Yaskawa INFORM job: DEMO_ROOF_UPPER_0625_3PAINT_59.JBI

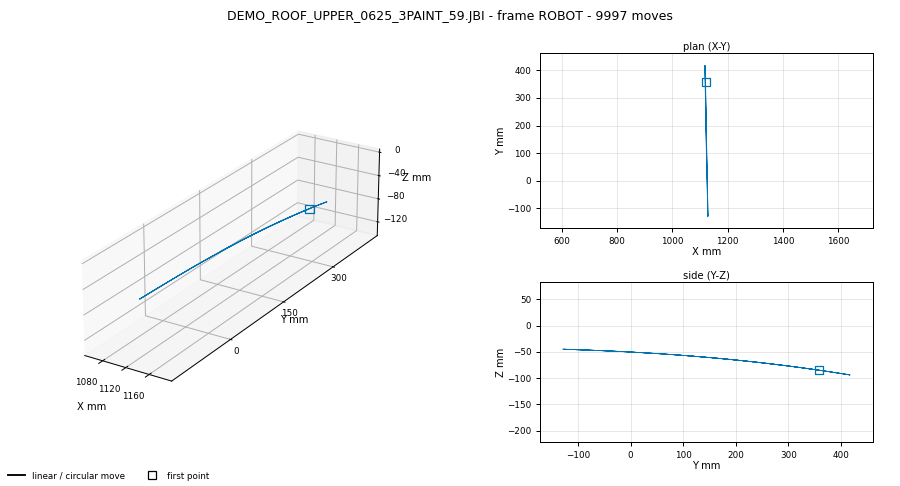
[picture p0: tool path of DEMO_ROOF_UPPER_0625_3PAINT_59.JBI in frame ROBOT, 9997 of 9997 moves have a stored position in this frame; points joined in program order, loops and branches not executed]
/JOB
//NAME DEMO_ROOF_UPPER_0625_3PAINT59
//POS
///NPOS 9997,0,0,0,0,0
///TOOL 0
///USER 0
///POSTYPE ROBOT
///RECTAN
///RCONF 1,0,0,0,0,0,0,0,0,0,0,0,0,0,0,0,0,0,0,0,0,0,0,0
C00000=1119.917,358.659,-84.729,-177.151,11.041,149.489
C00001=1119.921,358.412,-84.693,-177.154,11.038,149.489
C00002=1119.925,358.165,-84.658,-177.158,11.036,149.490
C00003=1119.929,357.918,-84.622,-177.161,11.033,149.490
C00004=1119.933,357.670,-84.586,-177.165,11.031,149.490
C00005=1119.936,357.423,-84.550,-177.168,11.029,149.490
C00006=1119.940,357.176,-84.514,-177.171,11.026,149.491
C00007=1119.944,356.928,-84.479,-177.175,11.024,149.491
C00008=1119.948,356.680,-84.443,-177.179,11.021,149.491
C00009=1119.952,356.433,-84.407,-177.182,11.019,149.491
C00010=1119.955,356.185,-84.372,-177.186,11.016,149.492
C00011=1119.959,355.938,-84.336,-177.189,11.014,149.492
C00012=1119.963,355.691,-84.301,-177.192,11.011,149.492
C00013=1119.967,355.444,-84.265,-177.196,11.009,149.492
C00014=1119.971,355.196,-84.229,-177.199,11.007,149.493
C00015=1119.975,354.948,-84.194,-177.203,11.004,149.493
C00016=1119.979,354.701,-84.158,-177.206,11.002,149.493
C00017=1119.982,354.453,-84.123,-177.209,10.999,149.493
C00018=1119.986,354.206,-84.087,-177.212,10.997,149.494
C00019=1119.990,353.959,-84.052,-177.217,10.994,149.494
C00020=1119.994,353.711,-84.016,-177.220,10.991,149.494
C00021=1119.997,353.464,-83.981,-177.223,10.989,149.494
C00022=1120.001,353.216,-83.945,-177.227,10.986,149.495
C00023=1120.006,352.969,-83.909,-177.230,10.984,149.495
C00024=1120.010,352.722,-83.874,-177.233,10.981,149.495
C00025=1120.013,352.474,-83.838,-177.237,10.979,149.495
C00026=1120.017,352.227,-83.803,-177.241,10.976,149.496
C00027=1120.021,351.979,-83.767,-177.244,10.974,149.496
C00028=1120.025,351.731,-83.732,-177.248,10.971,149.496
C00029=1120.029,351.484,-83.697,-177.251,10.969,149.496
C00030=1120.033,351.237,-83.662,-177.254,10.966,149.497
C00031=1120.036,350.989,-83.626,-177.258,10.964,149.497
C00032=1120.040,350.742,-83.591,-177.261,10.961,149.497
C00033=1120.045,350.494,-83.556,-177.265,10.958,149.497
C00034=1120.048,350.247,-83.521,-177.268,10.956,149.498
C00035=1120.052,349.999,-83.485,-177.272,10.953,149.498
C00036=1120.056,349.751,-83.450,-177.275,10.951,149.498
C00037=1120.059,349.505,-83.416,-177.279,10.948,149.498
C00038=1120.063,349.292,-83.385,-177.282,10.946,149.498
C00039=1120.066,349.080,-83.355,-177.284,10.944,149.499
C00040=1120.070,348.867,-83.325,-177.287,10.942,149.499
C00041=1120.073,348.655,-83.295,-177.290,10.940,149.499
C00042=1120.077,348.443,-83.265,-177.293,10.937,149.499
C00043=1120.079,348.230,-83.234,-177.296,10.935,149.499
C00044=1120.083,348.018,-83.204,-177.298,10.933,149.499
C00045=1120.086,347.805,-83.174,-177.301,10.931,149.500
C00046=1120.090,347.558,-83.139,-177.305,10.929,149.500
C00047=1120.095,347.310,-83.104,-177.307,10.926,149.500
C00048=1120.098,347.063,-83.069,-177.310,10.924,149.500
C00049=1120.101,346.815,-83.034,-177.313,10.922,149.500
C00050=1120.106,346.568,-82.999,-177.317,10.919,149.501
C00051=1120.110,346.320,-82.964,-177.320,10.917,149.501
C00052=1120.113,346.073,-82.929,-177.323,10.914,149.501
C00053=1120.118,345.825,-82.894,-177.327,10.912,149.501
C00054=1120.122,345.578,-82.859,-177.330,10.909,149.501
C00055=1120.125,345.331,-82.825,-177.333,10.907,149.502
C00056=1120.129,345.083,-82.789,-177.336,10.904,149.502
C00057=1120.133,344.835,-82.755,-177.340,10.902,149.502
C00058=1120.138,344.588,-82.720,-177.343,10.899,149.502
C00059=1120.141,344.340,-82.685,-177.346,10.897,149.503
C00060=1120.145,344.093,-82.651,-177.349,10.894,149.503
C00061=1120.149,343.846,-82.615,-177.352,10.891,149.503
C00062=1120.153,343.597,-82.580,-177.355,10.890,149.503
C00063=1120.157,343.350,-82.546,-177.358,10.887,149.503
C00064=1120.160,343.103,-82.511,-177.362,10.885,149.504
C00065=1120.165,342.855,-82.476,-177.365,10.882,149.504
C00066=1120.169,342.607,-82.442,-177.368,10.880,149.504
C00067=1120.173,342.360,-82.408,-177.371,10.877,149.504
C00068=1120.176,342.113,-82.372,-177.375,10.875,149.504
C00069=1120.180,341.865,-82.337,-177.378,10.872,149.505
C00070=1120.184,341.617,-82.304,-177.381,10.869,149.505
C00071=1120.188,341.369,-82.269,-177.384,10.867,149.505
C00072=1120.193,341.122,-82.234,-177.387,10.865,149.505
C00073=1120.195,340.875,-82.199,-177.391,10.862,149.505
C00074=1120.200,340.627,-82.165,-177.394,10.860,149.506
C00075=1120.204,340.379,-82.130,-177.397,10.857,149.506
C00076=1120.208,340.132,-82.096,-177.400,10.854,149.506
C00077=1120.212,339.884,-82.061,-177.403,10.853,149.506
C00078=1120.216,339.637,-82.027,-177.406,10.850,149.506
C00079=1120.220,339.389,-81.993,-177.410,10.848,149.507
C00080=1120.224,339.141,-81.958,-177.413,10.845,149.507
C00081=1120.227,338.894,-81.923,-177.416,10.843,149.507
C00082=1120.232,338.647,-81.889,-177.419,10.840,149.507
C00083=1120.235,338.399,-81.854,-177.422,10.838,149.507
C00084=1120.239,338.151,-81.820,-177.425,10.835,149.507
C00085=1120.243,337.904,-81.786,-177.429,10.832,149.508
C00086=1120.247,337.656,-81.751,-177.432,10.830,149.508
C00087=1120.251,337.409,-81.717,-177.435,10.827,149.508
C00088=1120.255,337.161,-81.683,-177.439,10.825,149.508
C00089=1120.259,336.914,-81.649,-177.442,10.822,149.508
C00090=1120.263,336.665,-81.615,-177.445,10.820,149.509
C00091=1120.267,336.418,-81.581,-177.448,10.818,149.509
C00092=1120.271,336.170,-81.546,-177.451,10.816,149.509
C00093=1120.275,335.923,-81.512,-177.454,10.813,149.509
C00094=1120.278,335.711,-81.482,-177.457,10.810,149.509
C00095=1120.282,335.498,-81.454,-177.459,10.808,149.509
C00096=1120.285,335.285,-81.424,-177.462,10.807,149.510
C00097=1120.289,335.073,-81.394,-177.465,10.804,149.510
C00098=1120.292,334.860,-81.365,-177.468,10.802,149.510
C00099=1120.295,334.648,-81.335,-177.471,10.800,149.510
C00100=1120.299,334.435,-81.306,-177.473,10.798,149.510
C00101=1120.302,334.223,-81.277,-177.476,10.796,149.510
C00102=1120.306,333.975,-81.243,-177.479,10.793,149.511
C00103=1120.310,333.727,-81.209,-177.482,10.791,149.511
C00104=1120.314,333.480,-81.175,-177.485,10.788,149.511
C00105=1120.318,333.233,-81.141,-177.488,10.786,149.511
C00106=1120.321,332.985,-81.107,-177.492,10.783,149.511
C00107=1120.326,332.737,-81.073,-177.495,10.781,149.512
C00108=1120.329,332.489,-81.039,-177.498,10.778,149.512
C00109=1120.333,332.242,-81.005,-177.501,10.776,149.512
C00110=1120.338,331.994,-80.971,-177.505,10.773,149.512
C00111=1120.341,331.746,-80.937,-177.508,10.771,149.512
C00112=1120.345,331.499,-80.903,-177.511,10.768,149.513
C00113=1120.350,331.251,-80.869,-177.514,10.766,149.513
C00114=1120.353,331.003,-80.835,-177.517,10.764,149.513
C00115=1120.357,330.755,-80.802,-177.520,10.761,149.513
C00116=1120.361,330.508,-80.768,-177.523,10.759,149.513
C00117=1120.366,330.261,-80.734,-177.526,10.756,149.514
C00118=1120.369,330.012,-80.700,-177.530,10.754,149.514
C00119=1120.373,329.765,-80.666,-177.533,10.751,149.514
C00120=1120.377,329.517,-80.633,-177.536,10.748,149.514
C00121=1120.381,329.269,-80.598,-177.539,10.746,149.514
C00122=1120.385,329.022,-80.565,-177.542,10.743,149.514
C00123=1120.389,328.774,-80.531,-177.546,10.741,149.515
C00124=1120.393,328.527,-80.498,-177.549,10.738,149.515
C00125=1120.397,328.279,-80.464,-177.552,10.736,149.515
C00126=1120.401,328.031,-80.430,-177.555,10.733,149.515
C00127=1120.406,327.783,-80.397,-177.558,10.731,149.516
C00128=1120.409,327.536,-80.363,-177.561,10.729,149.516
C00129=1120.413,327.288,-80.329,-177.564,10.726,149.516
C00130=1120.417,327.041,-80.296,-177.567,10.724,149.516
C00131=1120.421,326.793,-80.262,-177.571,10.721,149.516
C00132=1120.425,326.545,-80.229,-177.574,10.719,149.516
C00133=1120.429,326.297,-80.194,-177.577,10.716,149.517
C00134=1120.433,326.049,-80.161,-177.580,10.714,149.517
C00135=1120.437,325.801,-80.128,-177.583,10.711,149.517
C00136=1120.441,325.554,-80.094,-177.587,10.708,149.517
C00137=1120.445,325.307,-80.061,-177.590,10.706,149.517
C00138=1120.449,325.058,-80.028,-177.593,10.703,149.517
C00139=1120.453,324.810,-79.994,-177.596,10.701,149.518
C00140=1120.457,324.563,-79.961,-177.599,10.698,149.518
C00141=1120.461,324.316,-79.927,-177.602,10.696,149.518
C00142=1120.465,324.068,-79.894,-177.605,10.694,149.518
C00143=1120.469,323.820,-79.861,-177.608,10.691,149.519
C00144=1120.472,323.572,-79.827,-177.611,10.689,149.519
C00145=1120.477,323.325,-79.794,-177.615,10.686,149.519
C00146=1120.481,323.077,-79.761,-177.618,10.684,149.519
C00147=1120.485,322.829,-79.727,-177.621,10.681,149.519
C00148=1120.489,322.581,-79.694,-177.624,10.678,149.519
C00149=1120.493,322.334,-79.661,-177.628,10.676,149.520
C00150=1120.497,322.121,-79.632,-177.630,10.674,149.520
C00151=1120.499,321.908,-79.604,-177.633,10.671,149.520
C00152=1120.503,321.695,-79.575,-177.635,10.670,149.520
C00153=1120.507,321.483,-79.547,-177.638,10.668,149.520
C00154=1120.510,321.271,-79.518,-177.641,10.665,149.520
C00155=1120.513,321.058,-79.489,-177.643,10.663,149.521
C00156=1120.516,320.845,-79.461,-177.646,10.661,149.521
C00157=1120.521,320.632,-79.433,-177.649,10.659,149.521
C00158=1120.524,320.384,-79.400,-177.652,10.656,149.521
C00159=1120.528,320.136,-79.367,-177.655,10.654,149.521
C00160=1120.532,319.889,-79.333,-177.659,10.651,149.521
C00161=1120.536,319.641,-79.300,-177.661,10.648,149.522
C00162=1120.540,319.393,-79.268,-177.664,10.647,149.522
C00163=1120.544,319.146,-79.235,-177.668,10.644,149.522
C00164=1120.548,318.898,-79.201,-177.670,10.641,149.522
C00165=1120.552,318.650,-79.168,-177.674,10.639,149.522
C00166=1120.556,318.402,-79.135,-177.677,10.636,149.522
C00167=1120.561,318.155,-79.102,-177.680,10.634,149.523
C00168=1120.564,317.907,-79.069,-177.683,10.631,149.523
C00169=1120.568,317.659,-79.037,-177.686,10.629,149.523
C00170=1120.573,317.411,-79.004,-177.690,10.626,149.523
C00171=1120.577,317.164,-78.971,-177.693,10.624,149.524
C00172=1120.580,316.916,-78.938,-177.696,10.621,149.524
C00173=1120.584,316.668,-78.905,-177.699,10.618,149.524
C00174=1120.589,316.420,-78.872,-177.702,10.616,149.524
C00175=1120.593,316.172,-78.839,-177.705,10.614,149.524
C00176=1120.596,315.925,-78.807,-177.708,10.612,149.524
C00177=1120.600,315.677,-78.774,-177.711,10.609,149.525
C00178=1120.605,315.429,-78.741,-177.714,10.606,149.525
C00179=1120.609,315.181,-78.708,-177.717,10.604,149.525
C00180=1120.612,314.934,-78.675,-177.721,10.601,149.525
C00181=1120.617,314.685,-78.643,-177.724,10.599,149.525
C00182=1120.621,314.438,-78.610,-177.727,10.596,149.525
C00183=1120.624,314.190,-78.577,-177.730,10.593,149.526
C00184=1120.629,313.942,-78.545,-177.733,10.591,149.526
C00185=1120.633,313.694,-78.512,-177.736,10.588,149.526
C00186=1120.636,313.447,-78.479,-177.740,10.586,149.526
C00187=1120.641,313.198,-78.447,-177.742,10.584,149.526
C00188=1120.645,312.951,-78.414,-177.745,10.581,149.527
C00189=1120.649,312.703,-78.382,-177.748,10.579,149.527
C00190=1120.653,312.455,-78.349,-177.752,10.576,149.527
C00191=1120.657,312.206,-78.316,-177.755,10.573,149.527
C00192=1120.661,311.959,-78.284,-177.758,10.571,149.527
C00193=1120.666,311.711,-78.251,-177.761,10.569,149.528
C00194=1120.669,311.464,-78.219,-177.764,10.566,149.528
C00195=1120.673,311.216,-78.186,-177.768,10.563,149.528
C00196=1120.677,310.968,-78.154,-177.770,10.561,149.528
C00197=1120.681,310.720,-78.121,-177.774,10.558,149.528
C00198=1120.685,310.472,-78.088,-177.777,10.555,149.528
C00199=1120.689,310.224,-78.056,-177.779,10.554,149.529
C00200=1120.693,309.976,-78.023,-177.783,10.551,149.529
C00201=1120.697,309.728,-77.991,-177.786,10.548,149.529
C00202=1120.702,309.481,-77.959,-177.789,10.546,149.529
C00203=1120.705,309.233,-77.927,-177.792,10.543,149.529
C00204=1120.710,308.985,-77.894,-177.795,10.541,149.529
C00205=1120.714,308.737,-77.863,-177.798,10.538,149.530
C00206=1120.717,308.525,-77.835,-177.801,10.536,149.530
C00207=1120.721,308.311,-77.806,-177.804,10.534,149.530
C00208=1120.724,308.099,-77.779,-177.806,10.532,149.530
C00209=1120.728,307.886,-77.752,-177.809,10.530,149.530
C00210=1120.731,307.673,-77.724,-177.812,10.527,149.530
C00211=1120.735,307.460,-77.696,-177.814,10.525,149.531
C00212=1120.738,307.247,-77.668,-177.817,10.523,149.531
C00213=1120.742,307.035,-77.641,-177.820,10.521,149.531
C00214=1120.746,306.786,-77.608,-177.823,10.518,149.531
C00215=1120.750,306.538,-77.576,-177.826,10.516,149.531
C00216=1120.754,306.292,-77.544,-177.829,10.513,149.531
C00217=1120.758,306.043,-77.512,-177.832,10.510,149.532
C00218=1120.762,305.795,-77.480,-177.835,10.509,149.532
C00219=1120.766,305.547,-77.448,-177.838,10.506,149.532
C00220=1120.771,305.300,-77.416,-177.841,10.504,149.532
C00221=1120.774,305.052,-77.384,-177.844,10.501,149.532
C00222=1120.779,304.803,-77.352,-177.847,10.498,149.533
C00223=1120.782,304.556,-77.319,-177.850,10.496,149.533
C00224=1120.786,304.308,-77.288,-177.854,10.493,149.533
C00225=1120.791,304.060,-77.255,-177.857,10.491,149.533
C00226=1120.795,303.812,-77.223,-177.860,10.488,149.533
C00227=1120.798,303.564,-77.192,-177.863,10.485,149.533
C00228=1120.803,303.316,-77.160,-177.866,10.483,149.534
C00229=1120.807,303.068,-77.128,-177.870,10.480,149.534
C00230=1120.811,302.820,-77.096,-177.872,10.478,149.534
C00231=1120.816,302.573,-77.064,-177.875,10.476,149.534
C00232=1120.820,302.325,-77.032,-177.878,10.473,149.534
C00233=1120.823,302.077,-77.000,-177.881,10.471,149.535
C00234=1120.828,301.829,-76.969,-177.884,10.468,149.535
C00235=1120.832,301.581,-76.936,-177.888,10.465,149.535
C00236=1120.836,301.332,-76.905,-177.891,10.463,149.535
C00237=1120.840,301.085,-76.874,-177.894,10.460,149.535
C00238=1120.844,300.837,-76.842,-177.897,10.457,149.535
C00239=1120.848,300.588,-76.809,-177.900,10.455,149.536
C00240=1120.853,300.341,-76.778,-177.903,10.452,149.536
C00241=1120.856,300.093,-76.746,-177.906,10.451,149.536
C00242=1120.860,299.845,-76.714,-177.909,10.448,149.536
C00243=1120.865,299.597,-76.683,-177.912,10.445,149.536
C00244=1120.869,299.349,-76.651,-177.915,10.443,149.536
C00245=1120.873,299.101,-76.619,-177.918,10.440,149.537
C00246=1120.877,298.853,-76.588,-177.921,10.437,149.537
C00247=1120.881,298.605,-76.556,-177.925,10.435,149.537
C00248=1120.886,298.357,-76.525,-177.928,10.432,149.537
C00249=1120.889,298.109,-76.493,-177.931,10.430,149.537
C00250=1120.893,297.861,-76.461,-177.934,10.427,149.537
C00251=1120.897,297.614,-76.430,-177.937,10.425,149.538
C00252=1120.902,297.365,-76.398,-177.939,10.423,149.538
C00253=1120.906,297.118,-76.367,-177.943,10.420,149.538
C00254=1120.910,296.870,-76.335,-177.946,10.417,149.538
C00255=1120.915,296.622,-76.304,-177.949,10.415,149.538
C00256=1120.918,296.374,-76.272,-177.952,10.412,149.539
C00257=1120.922,296.125,-76.241,-177.955,10.410,149.539
C00258=1120.927,295.878,-76.210,-177.958,10.407,149.539
C00259=1120.930,295.630,-76.178,-177.962,10.405,149.539
C00260=1120.935,295.382,-76.147,-177.965,10.402,149.539
C00261=1120.939,295.134,-76.115,-177.968,10.399,149.539
C00262=1120.943,294.920,-76.089,-177.970,10.397,149.540
C00263=1120.946,294.708,-76.061,-177.973,10.396,149.540
C00264=1120.949,294.495,-76.035,-177.975,10.393,149.540
C00265=1120.953,294.282,-76.008,-177.978,10.391,149.540
C00266=1120.957,294.069,-75.981,-177.980,10.389,149.540
C00267=1120.960,293.856,-75.954,-177.983,10.386,149.540
C00268=1120.964,293.643,-75.927,-177.986,10.384,149.540
C00269=1120.968,293.430,-75.900,-177.988,10.383,149.541
C00270=1120.972,293.181,-75.869,-177.991,10.380,149.541
C00271=1120.975,292.934,-75.838,-177.995,10.378,149.541
C00272=1120.979,292.686,-75.807,-177.998,10.375,149.541
C00273=1120.983,292.438,-75.776,-178.001,10.372,149.541
C00274=1120.987,292.190,-75.744,-178.004,10.370,149.542
C00275=1120.992,291.942,-75.714,-178.007,10.367,149.542
C00276=1120.996,291.694,-75.682,-178.010,10.364,149.542
C00277=1121.000,291.446,-75.651,-178.013,10.362,149.542
C00278=1121.004,291.198,-75.619,-178.016,10.359,149.542
C00279=1121.008,290.950,-75.589,-178.019,10.357,149.542
C00280=1121.012,290.701,-75.558,-178.022,10.355,149.543
C00281=1121.017,290.454,-75.527,-178.025,10.352,149.543
C00282=1121.020,290.205,-75.495,-178.028,10.350,149.543
C00283=1121.025,289.958,-75.464,-178.031,10.347,149.543
C00284=1121.030,289.710,-75.434,-178.035,10.344,149.543
C00285=1121.032,289.462,-75.402,-178.038,10.342,149.543
C00286=1121.037,289.214,-75.372,-178.041,10.339,149.544
C00287=1121.041,288.965,-75.341,-178.044,10.336,149.544
C00288=1121.046,288.717,-75.310,-178.046,10.334,149.544
C00289=1121.050,288.469,-75.279,-178.049,10.332,149.544
C00290=1121.053,288.222,-75.248,-178.052,10.329,149.544
C00291=1121.058,287.974,-75.217,-178.056,10.327,149.545
C00292=1121.062,287.725,-75.186,-178.059,10.324,149.545
C00293=1121.067,287.477,-75.155,-178.062,10.322,149.545
C00294=1121.070,287.229,-75.125,-178.065,10.319,149.545
C00295=1121.074,286.981,-75.094,-178.068,10.316,149.545
C00296=1121.079,286.733,-75.063,-178.071,10.314,149.545
C00297=1121.083,286.485,-75.033,-178.074,10.311,149.545
C00298=1121.087,286.236,-75.002,-178.077,10.309,149.546
C00299=1121.091,285.989,-74.970,-178.080,10.307,149.546
C00300=1121.095,285.741,-74.940,-178.083,10.304,149.546
C00301=1121.099,285.493,-74.909,-178.086,10.301,149.546
C00302=1121.104,285.245,-74.878,-178.089,10.299,149.547
C00303=1121.108,284.997,-74.848,-178.092,10.296,149.547
C00304=1121.112,284.749,-74.817,-178.095,10.293,149.547
C00305=1121.116,284.501,-74.786,-178.099,10.291,149.547
C00306=1121.120,284.253,-74.756,-178.102,10.288,149.547
C00307=1121.124,284.004,-74.726,-178.104,10.287,149.547
C00308=1121.129,283.756,-74.695,-178.107,10.284,149.547
C00309=1121.133,283.508,-74.665,-178.111,10.281,149.548
C00310=1121.137,283.259,-74.634,-178.113,10.279,149.548
C00311=1121.141,283.012,-74.603,-178.116,10.276,149.548
C00312=1121.145,282.764,-74.573,-178.120,10.273,149.548
C00313=1121.149,282.516,-74.542,-178.123,10.271,149.548
C00314=1121.153,282.267,-74.511,-178.126,10.268,149.549
C00315=1121.158,282.019,-74.481,-178.129,10.266,149.549
C00316=1121.162,281.771,-74.451,-178.132,10.263,149.549
C00317=1121.167,281.523,-74.420,-178.135,10.261,149.549
C00318=1121.172,281.148,-74.374,-178.140,10.256,149.549
C00319=1121.179,280.772,-74.328,-178.145,10.253,149.550
C00320=1121.185,280.397,-74.283,-178.150,10.248,149.550
C00321=1121.192,280.022,-74.236,-178.155,10.244,149.550
C00322=1121.196,279.774,-74.207,-178.158,10.242,149.550
C00323=1121.201,279.526,-74.176,-178.161,10.239,149.551
C00324=1121.204,279.277,-74.145,-178.164,10.236,149.551
C00325=1121.209,279.029,-74.115,-178.168,10.233,149.551
C00326=1121.213,278.781,-74.085,-178.171,10.231,149.551
C00327=1121.216,278.534,-74.055,-178.174,10.228,149.551
C00328=1121.221,278.285,-74.025,-178.178,10.225,149.552
C00329=1121.225,278.037,-73.995,-178.181,10.223,149.552
C00330=1121.230,277.788,-73.964,-178.184,10.220,149.552
C00331=1121.233,277.540,-73.934,-178.187,10.217,149.552
C00332=1121.237,277.293,-73.904,-178.190,10.215,149.552
C00333=1121.242,277.044,-73.874,-178.194,10.211,149.552
C00334=1121.246,276.797,-73.844,-178.197,10.209,149.553
C00335=1121.250,276.548,-73.814,-178.200,10.206,149.553
C00336=1121.254,276.300,-73.783,-178.203,10.203,149.553
C00337=1121.259,276.051,-73.754,-178.206,10.201,149.553
C00338=1121.262,275.804,-73.724,-178.209,10.198,149.553
C00339=1121.267,275.555,-73.694,-178.212,10.195,149.553
C00340=1121.272,275.307,-73.664,-178.215,10.192,149.553
C00341=1121.275,275.059,-73.634,-178.218,10.190,149.554
C00342=1121.280,274.811,-73.605,-178.221,10.187,149.554
C00343=1121.284,274.563,-73.574,-178.224,10.185,149.554
C00344=1121.288,274.315,-73.544,-178.227,10.182,149.554
C00345=1121.292,274.066,-73.515,-178.230,10.179,149.554
C00346=1121.296,273.818,-73.484,-178.233,10.177,149.554
C00347=1121.301,273.570,-73.454,-178.236,10.174,149.554
C00348=1121.305,273.321,-73.425,-178.239,10.171,149.554
C00349=1121.309,273.074,-73.395,-178.242,10.168,149.555
C00350=1121.313,272.825,-73.365,-178.244,10.166,149.555
C00351=1121.317,272.577,-73.336,-178.247,10.164,149.555
C00352=1121.322,272.329,-73.305,-178.250,10.161,149.555
C00353=1121.326,272.081,-73.276,-178.253,10.158,149.555
C00354=1121.330,271.833,-73.246,-178.256,10.155,149.555
C00355=1121.334,271.584,-73.217,-178.259,10.153,149.555
C00356=1121.338,271.337,-73.187,-178.262,10.150,149.555
C00357=1121.342,271.088,-73.157,-178.265,10.148,149.556
C00358=1121.348,270.789,-73.121,-178.268,10.145,149.556
C00359=1121.353,270.490,-73.086,-178.272,10.141,149.556
C00360=1121.358,270.191,-73.049,-178.275,10.138,149.556
C00361=1121.363,269.892,-73.014,-178.278,10.135,149.556
C00362=1121.367,269.643,-72.985,-178.281,10.133,149.556
C00363=1121.371,269.395,-72.955,-178.283,10.130,149.556
C00364=1121.375,269.147,-72.926,-178.286,10.127,149.556
C00365=1121.380,268.899,-72.896,-178.289,10.125,149.556
C00366=1121.383,268.651,-72.866,-178.292,10.123,149.556
C00367=1121.388,268.402,-72.836,-178.295,10.120,149.557
C00368=1121.392,268.154,-72.807,-178.298,10.117,149.557
C00369=1121.397,267.907,-72.778,-178.300,10.115,149.557
C00370=1121.401,267.693,-72.752,-178.302,10.113,149.557
C00371=1121.404,267.480,-72.727,-178.305,10.110,149.557
C00372=1121.408,267.266,-72.702,-178.307,10.108,149.557
C00373=1121.412,267.053,-72.677,-178.310,10.106,149.557
C00374=1121.415,266.839,-72.652,-178.312,10.104,149.557
C00375=1121.418,266.627,-72.626,-178.314,10.102,149.557
C00376=1121.423,266.414,-72.601,-178.316,10.100,149.557
C00377=1121.426,266.201,-72.576,-178.319,10.098,149.558
C00378=1121.430,265.952,-72.546,-178.321,10.095,149.558
C00379=1121.434,265.704,-72.517,-178.324,10.093,149.558
C00380=1121.439,265.456,-72.487,-178.327,10.091,149.558
C00381=1121.443,265.207,-72.458,-178.329,10.089,149.558
C00382=1121.447,264.959,-72.429,-178.332,10.086,149.558
C00383=1121.451,264.710,-72.400,-178.334,10.083,149.558
C00384=1121.456,264.462,-72.370,-178.337,10.081,149.558
C00385=1121.460,264.214,-72.341,-178.340,10.078,149.559
C00386=1121.465,263.966,-72.312,-178.344,10.075,149.559
C00387=1121.469,263.718,-72.282,-178.347,10.072,149.559
C00388=1121.473,263.469,-72.254,-178.351,10.069,149.559
C00389=1121.477,263.221,-72.225,-178.354,10.066,149.559
C00390=1121.481,262.973,-72.195,-178.358,10.063,149.560
C00391=1121.486,262.725,-72.166,-178.361,10.061,149.560
C00392=1121.490,262.476,-72.137,-178.365,10.057,149.560
C00393=1121.494,262.228,-72.108,-178.368,10.055,149.560
C00394=1121.499,261.980,-72.079,-178.371,10.052,149.560
C00395=1121.502,261.732,-72.050,-178.375,10.049,149.560
C00396=1121.506,261.483,-72.021,-178.378,10.046,149.561
C00397=1121.511,261.235,-71.992,-178.381,10.043,149.561
C00398=1121.515,260.987,-71.962,-178.384,10.040,149.561
C00399=1121.520,260.738,-71.934,-178.388,10.037,149.561
C00400=1121.523,260.490,-71.905,-178.391,10.034,149.561
C00401=1121.528,260.242,-71.876,-178.394,10.031,149.561
C00402=1121.533,259.994,-71.847,-178.397,10.028,149.561
C00403=1121.537,259.746,-71.818,-178.400,10.025,149.561
C00404=1121.541,259.497,-71.789,-178.403,10.023,149.562
C00405=1121.545,259.249,-71.760,-178.406,10.020,149.562
C00406=1121.550,259.001,-71.732,-178.409,10.016,149.562
C00407=1121.553,258.753,-71.703,-178.412,10.014,149.562
C00408=1121.558,258.504,-71.674,-178.415,10.011,149.562
C00409=1121.563,258.256,-71.645,-178.418,10.008,149.562
C00410=1121.567,258.007,-71.616,-178.421,10.005,149.562
C00411=1121.570,257.759,-71.587,-178.424,10.003,149.562
C00412=1121.575,257.510,-71.559,-178.427,10.000,149.562
C00413=1121.580,257.263,-71.529,-178.430,9.997,149.562
C00414=1121.584,257.014,-71.501,-178.433,9.994,149.562
C00415=1121.588,256.765,-71.473,-178.435,9.991,149.563
C00416=1121.592,256.518,-71.444,-178.438,9.988,149.563
C00417=1121.597,256.269,-71.415,-178.441,9.986,149.563
C00418=1121.601,256.020,-71.387,-178.444,9.983,149.563
C00419=1121.605,255.773,-71.358,-178.445,9.981,149.563
C00420=1121.610,255.524,-71.329,-178.445,9.980,149.562
C00421=1121.613,255.276,-71.300,-178.446,9.978,149.562
C00422=1121.618,255.028,-71.272,-178.447,9.977,149.562
C00423=1121.623,254.779,-71.243,-178.448,9.975,149.562
C00424=1121.626,254.531,-71.215,-178.449,9.974,149.562
C00425=1121.631,254.283,-71.186,-178.450,9.972,149.562
C00426=1121.635,254.069,-71.162,-178.451,9.971,149.562
C00427=1121.638,253.856,-71.137,-178.453,9.969,149.562
C00428=1121.642,253.643,-71.113,-178.455,9.967,149.562
C00429=1121.646,253.429,-71.088,-178.456,9.966,149.562
C00430=1121.649,253.216,-71.063,-178.459,9.964,149.562
C00431=1121.653,253.003,-71.039,-178.460,9.962,149.562
C00432=1121.657,252.789,-71.014,-178.462,9.960,149.562
C00433=1121.660,252.576,-70.990,-178.465,9.958,149.562
C00434=1121.665,252.327,-70.962,-178.467,9.956,149.562
C00435=1121.668,252.079,-70.933,-178.470,9.954,149.563
C00436=1121.673,251.831,-70.904,-178.473,9.951,149.563
C00437=1121.677,251.583,-70.876,-178.476,9.948,149.563
C00438=1121.682,251.334,-70.848,-178.479,9.946,149.563
C00439=1121.686,251.086,-70.820,-178.483,9.943,149.563
C00440=1121.690,250.838,-70.790,-178.487,9.939,149.564
C00441=1121.694,250.589,-70.762,-178.490,9.937,149.564
C00442=1121.699,250.341,-70.734,-178.494,9.933,149.564
C00443=1121.703,250.092,-70.706,-178.499,9.930,149.565
C00444=1121.708,249.844,-70.677,-178.503,9.927,149.565
C00445=1121.712,249.595,-70.649,-178.508,9.923,149.565
C00446=1121.716,249.348,-70.621,-178.512,9.920,149.565
C00447=1121.720,249.099,-70.593,-178.517,9.916,149.566
C00448=1121.724,248.850,-70.565,-178.522,9.911,149.566
C00449=1121.729,248.602,-70.537,-178.527,9.907,149.566
C00450=1121.733,248.353,-70.508,-178.533,9.903,149.567
C00451=1121.737,248.106,-70.480,-178.537,9.899,149.567
C00452=1121.741,247.857,-70.452,-178.543,9.895,149.568
C00453=1121.746,247.609,-70.424,-178.549,9.890,149.568
C00454=1121.750,247.360,-70.396,-178.553,9.886,149.568
C00455=1121.755,247.112,-70.369,-178.554,9.883,149.568
C00456=1121.759,246.863,-70.340,-178.556,9.881,149.568
C00457=1121.764,246.615,-70.312,-178.558,9.879,149.568
C00458=1121.768,246.367,-70.284,-178.560,9.876,149.568
C00459=1121.772,246.118,-70.256,-178.561,9.874,149.568
C00460=1121.777,245.870,-70.228,-178.563,9.872,149.567
C00461=1121.781,245.621,-70.200,-178.565,9.870,149.567
C00462=1121.785,245.373,-70.173,-178.566,9.867,149.567
C00463=1121.789,245.125,-70.144,-178.568,9.865,149.567
C00464=1121.794,244.876,-70.116,-178.570,9.863,149.567
C00465=1121.798,244.627,-70.089,-178.572,9.860,149.567
C00466=1121.802,244.379,-70.061,-178.574,9.858,149.567
C00467=1121.807,244.132,-70.033,-178.576,9.856,149.567
C00468=1121.810,243.883,-70.005,-178.578,9.853,149.567
C00469=1121.816,243.634,-69.977,-178.580,9.850,149.567
C00470=1121.820,243.386,-69.949,-178.582,9.848,149.567
C00471=1121.824,243.138,-69.921,-178.584,9.846,149.567
C00472=1121.828,242.888,-69.894,-178.586,9.844,149.567
C00473=1121.832,242.641,-69.866,-178.588,9.841,149.567
C00474=1121.837,242.393,-69.838,-178.591,9.838,149.567
C00475=1121.841,242.143,-69.810,-178.593,9.836,149.567
C00476=1121.846,241.895,-69.783,-178.595,9.834,149.567
C00477=1121.850,241.647,-69.754,-178.597,9.832,149.567
C00478=1121.854,241.398,-69.727,-178.600,9.829,149.567
C00479=1121.859,241.150,-69.700,-178.602,9.826,149.567
C00480=1121.863,240.901,-69.672,-178.604,9.824,149.567
C00481=1121.867,240.653,-69.644,-178.607,9.821,149.567
C00482=1121.871,240.440,-69.620,-178.609,9.819,149.567
C00483=1121.875,240.226,-69.596,-178.611,9.817,149.567
C00484=1121.878,240.013,-69.573,-178.613,9.815,149.567
C00485=1121.881,239.799,-69.549,-178.615,9.813,149.567
C00486=1121.886,239.586,-69.526,-178.617,9.811,149.567
C00487=1121.889,239.372,-69.502,-178.619,9.808,149.567
C00488=1121.893,239.159,-69.478,-178.622,9.806,149.567
C00489=1121.897,238.946,-69.455,-178.624,9.804,149.567
C00490=1121.902,238.696,-69.427,-178.626,9.802,149.567
C00491=1121.906,238.448,-69.399,-178.629,9.799,149.568
C00492=1121.911,238.200,-69.372,-178.631,9.797,149.567
C00493=1121.914,237.951,-69.344,-178.634,9.794,149.568
C00494=1121.919,237.703,-69.317,-178.637,9.792,149.568
C00495=1121.923,237.455,-69.289,-178.639,9.790,149.568
C00496=1121.927,237.206,-69.261,-178.642,9.787,149.568
C00497=1121.932,236.957,-69.234,-178.644,9.784,149.568
C00498=1121.936,236.709,-69.207,-178.647,9.781,149.568
C00499=1121.941,236.461,-69.180,-178.650,9.779,149.568
C00500=1121.945,236.212,-69.151,-178.653,9.776,149.568
C00501=1121.949,235.964,-69.125,-178.655,9.774,149.568
C00502=1121.953,235.716,-69.098,-178.658,9.771,149.569
C00503=1121.957,235.467,-69.070,-178.661,9.768,149.569
C00504=1121.962,235.219,-69.043,-178.664,9.765,149.569
C00505=1121.967,234.970,-69.016,-178.667,9.762,149.569
C00506=1121.971,234.722,-68.989,-178.670,9.759,149.569
C00507=1121.975,234.473,-68.960,-178.673,9.757,149.569
C00508=1121.980,234.224,-68.933,-178.676,9.754,149.569
C00509=1121.984,233.976,-68.906,-178.679,9.751,149.569
C00510=1121.989,233.727,-68.879,-178.682,9.748,149.569
C00511=1121.993,233.480,-68.852,-178.685,9.746,149.569
C00512=1121.997,233.231,-68.825,-178.687,9.743,149.570
C00513=1122.001,232.982,-68.798,-178.691,9.739,149.570
C00514=1122.006,232.734,-68.771,-178.694,9.737,149.570
C00515=1122.011,232.485,-68.743,-178.697,9.734,149.570
C00516=1122.014,232.237,-68.715,-178.700,9.731,149.570
C00517=1122.018,231.988,-68.689,-178.703,9.728,149.570
C00518=1122.023,231.740,-68.662,-178.706,9.725,149.570
C00519=1122.028,231.491,-68.635,-178.709,9.722,149.570
C00520=1122.032,231.243,-68.608,-178.713,9.719,149.571
C00521=1122.037,230.994,-68.581,-178.716,9.716,149.571
C00522=1122.040,230.746,-68.554,-178.719,9.712,149.571
C00523=1122.045,230.497,-68.527,-178.722,9.710,149.571
C00524=1122.049,230.249,-68.500,-178.726,9.706,149.571
C00525=1122.054,230.000,-68.473,-178.730,9.703,149.571
C00526=1122.058,229.752,-68.446,-178.733,9.700,149.571
C00527=1122.063,229.503,-68.419,-178.736,9.696,149.571
C00528=1122.067,229.255,-68.392,-178.739,9.694,149.572
C00529=1122.071,229.007,-68.366,-178.743,9.690,149.572
C00530=1122.076,228.758,-68.338,-178.746,9.687,149.572
C00531=1122.080,228.509,-68.311,-178.749,9.683,149.572
C00532=1122.084,228.261,-68.285,-178.752,9.680,149.572
C00533=1122.089,228.012,-68.258,-178.755,9.677,149.572
C00534=1122.094,227.763,-68.231,-178.759,9.674,149.572
C00535=1122.097,227.515,-68.205,-178.761,9.671,149.572
C00536=1122.102,227.267,-68.178,-178.765,9.667,149.572
C00537=1122.106,227.018,-68.151,-178.768,9.664,149.572
C00538=1122.110,226.805,-68.128,-178.770,9.661,149.572
C00539=1122.114,226.591,-68.106,-178.773,9.658,149.572
C00540=1122.118,226.377,-68.082,-178.776,9.655,149.572
C00541=1122.121,226.164,-68.059,-178.778,9.652,149.572
C00542=1122.125,225.950,-68.036,-178.781,9.649,149.572
C00543=1122.129,225.736,-68.013,-178.783,9.647,149.572
C00544=1122.133,225.523,-67.991,-178.786,9.644,149.572
C00545=1122.137,225.309,-67.968,-178.789,9.641,149.572
C00546=1122.141,225.061,-67.941,-178.791,9.638,149.572
C00547=1122.145,224.813,-67.915,-178.794,9.634,149.572
C00548=1122.150,224.564,-67.888,-178.797,9.632,149.572
C00549=1122.154,224.315,-67.862,-178.800,9.628,149.572
C00550=1122.159,224.067,-67.835,-178.802,9.625,149.572
C00551=1122.163,223.818,-67.809,-178.806,9.622,149.572
C00552=1122.168,223.570,-67.782,-178.809,9.619,149.572
C00553=1122.172,223.321,-67.756,-178.811,9.616,149.572
C00554=1122.177,223.072,-67.729,-178.814,9.612,149.572
C00555=1122.180,222.824,-67.703,-178.817,9.609,149.572
C00556=1122.185,222.575,-67.677,-178.819,9.605,149.572
C00557=1122.189,222.327,-67.650,-178.822,9.602,149.572
C00558=1122.194,222.078,-67.624,-178.824,9.599,149.572
C00559=1122.198,221.830,-67.597,-178.827,9.596,149.572
C00560=1122.202,221.581,-67.571,-178.829,9.593,149.572
C00561=1122.207,221.332,-67.544,-178.832,9.590,149.572
C00562=1122.211,221.083,-67.519,-178.834,9.587,149.572
C00563=1122.216,220.835,-67.492,-178.837,9.584,149.571
C00564=1122.220,220.586,-67.466,-178.840,9.581,149.571
C00565=1122.224,220.337,-67.440,-178.842,9.577,149.571
C00566=1122.230,220.090,-67.413,-178.845,9.574,149.571
C00567=1122.234,219.841,-67.388,-178.847,9.571,149.571
C00568=1122.238,219.593,-67.361,-178.850,9.568,149.571
C00569=1122.243,219.343,-67.335,-178.852,9.565,149.571
C00570=1122.247,219.095,-67.309,-178.854,9.562,149.571
C00571=1122.251,218.846,-67.283,-178.857,9.558,149.571
C00572=1122.255,218.598,-67.257,-178.859,9.556,149.571
C00573=1122.260,218.349,-67.230,-178.861,9.553,149.571
C00574=1122.264,218.100,-67.204,-178.864,9.550,149.571
C00575=1122.269,217.852,-67.179,-178.866,9.546,149.570
C00576=1122.274,217.603,-67.152,-178.868,9.543,149.570
C00577=1122.278,217.355,-67.126,-178.870,9.541,149.570
C00578=1122.282,217.106,-67.100,-178.872,9.538,149.570
C00579=1122.286,216.857,-67.074,-178.875,9.534,149.570
C00580=1122.291,216.609,-67.047,-178.877,9.532,149.570
C00581=1122.296,216.361,-67.022,-178.879,9.529,149.570
C00582=1122.300,216.112,-66.996,-178.881,9.526,149.570
C00583=1122.304,215.863,-66.970,-178.883,9.523,149.570
C00584=1122.308,215.614,-66.945,-178.886,9.520,149.569
C00585=1122.313,215.366,-66.918,-178.887,9.517,149.569
C00586=1122.318,215.118,-66.892,-178.890,9.514,149.569
C00587=1122.322,214.869,-66.866,-178.891,9.512,149.569
C00588=1122.326,214.620,-66.841,-178.894,9.508,149.569
C00589=1122.331,214.371,-66.815,-178.896,9.506,149.569
C00590=1122.335,214.123,-66.789,-178.897,9.503,149.569
C00591=1122.340,213.875,-66.763,-178.900,9.500,149.568
C00592=1122.344,213.626,-66.737,-178.901,9.498,149.568
C00593=1122.348,213.377,-66.711,-178.903,9.495,149.568
C00594=1122.352,213.163,-66.690,-178.905,9.493,149.568
C00595=1122.356,212.950,-66.667,-178.907,9.491,149.568
C00596=1122.360,212.736,-66.645,-178.908,9.488,149.568
C00597=1122.364,212.522,-66.622,-178.910,9.486,149.568
C00598=1122.367,212.309,-66.600,-178.912,9.483,149.568
C00599=1122.371,212.094,-66.578,-178.914,9.481,149.568
C00600=1122.375,211.881,-66.556,-178.916,9.479,149.568
C00601=1122.379,211.667,-66.534,-178.918,9.475,149.568
C00602=1122.384,211.419,-66.509,-178.920,9.473,149.568
C00603=1122.388,211.170,-66.483,-178.923,9.470,149.568
C00604=1122.392,210.921,-66.457,-178.925,9.468,149.567
C00605=1122.397,210.672,-66.431,-178.927,9.465,149.567
C00606=1122.401,210.424,-66.406,-178.930,9.462,149.568
C00607=1122.406,210.175,-66.380,-178.932,9.460,149.567
C00608=1122.410,209.926,-66.354,-178.935,9.456,149.567
C00609=1122.415,209.678,-66.329,-178.937,9.454,149.567
C00610=1122.419,209.430,-66.303,-178.940,9.451,149.568
C00611=1122.423,209.181,-66.278,-178.942,9.448,149.567
C00612=1122.428,208.933,-66.252,-178.945,9.445,149.567
C00613=1122.432,208.684,-66.226,-178.947,9.443,149.568
C00614=1122.437,208.434,-66.201,-178.949,9.440,149.568
C00615=1122.442,208.186,-66.176,-178.952,9.437,149.568
C00616=1122.446,207.938,-66.150,-178.955,9.434,149.568
C00617=1122.450,207.689,-66.124,-178.958,9.431,149.568
C00618=1122.455,207.441,-66.099,-178.960,9.429,149.568
C00619=1122.459,207.192,-66.073,-178.963,9.426,149.568
C00620=1122.464,206.942,-66.048,-178.965,9.423,149.568
C00621=1122.468,206.694,-66.023,-178.968,9.421,149.568
C00622=1122.473,206.445,-65.997,-178.971,9.418,149.568
C00623=1122.477,206.197,-65.971,-178.974,9.415,149.568
C00624=1122.482,205.948,-65.947,-178.977,9.412,149.568
C00625=1122.486,205.699,-65.921,-178.980,9.409,149.568
C00626=1122.491,205.451,-65.896,-178.982,9.406,149.568
C00627=1122.495,205.203,-65.870,-178.985,9.403,149.568
C00628=1122.499,204.953,-65.845,-178.988,9.401,149.569
C00629=1122.504,204.705,-65.820,-178.990,9.397,149.568
C00630=1122.508,204.456,-65.794,-178.993,9.395,149.569
C00631=1122.513,204.207,-65.770,-178.996,9.392,149.569
C00632=1122.517,203.959,-65.744,-178.999,9.389,149.569
C00633=1122.523,203.710,-65.719,-179.003,9.386,149.569
C00634=1122.526,203.461,-65.694,-179.005,9.383,149.569
C00635=1122.530,203.213,-65.668,-179.008,9.380,149.569
C00636=1122.535,202.964,-65.644,-179.011,9.377,149.569
C00637=1122.540,202.715,-65.618,-179.015,9.374,149.569
C00638=1122.545,202.466,-65.593,-179.018,9.371,149.570
C00639=1122.548,202.218,-65.568,-179.021,9.368,149.570
C00640=1122.553,201.969,-65.543,-179.024,9.364,149.570
C00641=1122.558,201.720,-65.518,-179.027,9.362,149.570
C00642=1122.563,201.472,-65.493,-179.030,9.359,149.570
C00643=1122.566,201.223,-65.468,-179.033,9.355,149.570
C00644=1122.571,200.974,-65.443,-179.036,9.353,149.570
C00645=1122.576,200.726,-65.417,-179.040,9.349,149.570
C00646=1122.580,200.477,-65.393,-179.043,9.346,149.571
C00647=1122.585,200.228,-65.368,-179.046,9.342,149.570
C00648=1122.589,199.980,-65.343,-179.049,9.340,149.571
C00649=1122.593,199.731,-65.318,-179.053,9.336,149.571
C00650=1122.597,199.517,-65.297,-179.056,9.333,149.571
C00651=1122.602,199.303,-65.275,-179.059,9.331,149.571
C00652=1122.605,199.089,-65.254,-179.061,9.328,149.571
C00653=1122.609,198.875,-65.232,-179.064,9.325,149.571
C00654=1122.613,198.661,-65.211,-179.067,9.322,149.571
C00655=1122.617,198.448,-65.190,-179.070,9.319,149.571
C00656=1122.620,198.234,-65.168,-179.072,9.316,149.571
C00657=1122.624,198.019,-65.147,-179.075,9.313,149.572
C00658=1122.629,197.771,-65.122,-179.079,9.310,149.571
C00659=1122.633,197.522,-65.098,-179.082,9.306,149.572
C00660=1122.638,197.273,-65.073,-179.086,9.303,149.572
C00661=1122.642,197.025,-65.049,-179.089,9.299,149.572
C00662=1122.647,196.776,-65.024,-179.092,9.295,149.572
C00663=1122.651,196.528,-64.999,-179.096,9.292,149.572
C00664=1122.656,196.279,-64.974,-179.100,9.288,149.572
C00665=1122.660,196.030,-64.950,-179.101,9.285,149.572
C00666=1122.665,195.781,-64.925,-179.103,9.283,149.572
C00667=1122.669,195.532,-64.901,-179.104,9.280,149.572
C00668=1122.674,195.283,-64.876,-179.106,9.278,149.571
C00669=1122.678,195.035,-64.852,-179.108,9.275,149.571
C00670=1122.683,194.786,-64.826,-179.109,9.273,149.571
C00671=1122.687,194.538,-64.802,-179.111,9.270,149.571
C00672=1122.692,194.289,-64.778,-179.113,9.267,149.571
C00673=1122.696,194.040,-64.753,-179.115,9.265,149.571
C00674=1122.701,193.791,-64.729,-179.117,9.262,149.571
C00675=1122.705,193.543,-64.704,-179.119,9.260,149.571
C00676=1122.710,193.293,-64.679,-179.121,9.256,149.570
C00677=1122.714,193.045,-64.655,-179.123,9.254,149.570
C00678=1122.719,192.797,-64.631,-179.124,9.251,149.570
C00679=1122.723,192.547,-64.606,-179.126,9.249,149.570
C00680=1122.728,192.299,-64.582,-179.129,9.246,149.570
C00681=1122.733,192.050,-64.557,-179.130,9.243,149.570
C00682=1122.737,191.802,-64.533,-179.132,9.241,149.570
C00683=1122.741,191.552,-64.509,-179.135,9.238,149.570
C00684=1122.746,191.304,-64.484,-179.137,9.235,149.570
C00685=1122.751,191.055,-64.460,-179.139,9.232,149.570
C00686=1122.755,190.806,-64.435,-179.141,9.230,149.569
C00687=1122.760,190.557,-64.412,-179.143,9.227,149.569
C00688=1122.764,190.308,-64.388,-179.145,9.224,149.569
C00689=1122.769,190.060,-64.363,-179.147,9.222,149.569
C00690=1122.773,189.811,-64.339,-179.149,9.219,149.569
C00691=1122.777,189.562,-64.315,-179.151,9.216,149.569
C00692=1122.783,189.314,-64.290,-179.154,9.213,149.569
C00693=1122.787,189.065,-64.266,-179.156,9.211,149.569
C00694=1122.791,188.815,-64.242,-179.158,9.208,149.569
C00695=1122.796,188.567,-64.217,-179.161,9.205,149.569
C00696=1122.801,188.318,-64.193,-179.163,9.202,149.569
C00697=1122.805,188.070,-64.169,-179.165,9.199,149.569
C00698=1122.810,187.821,-64.145,-179.167,9.197,149.569
C00699=1122.814,187.571,-64.121,-179.170,9.194,149.569
C00700=1122.819,187.323,-64.097,-179.172,9.191,149.569
C00701=1122.823,187.075,-64.073,-179.174,9.188,149.569
C00702=1122.828,186.826,-64.048,-179.177,9.185,149.569
C00703=1122.833,186.577,-64.025,-179.179,9.182,149.569
C00704=1122.837,186.328,-64.000,-179.182,9.179,149.569
C00705=1122.841,186.079,-63.976,-179.184,9.177,149.569
C00706=1122.846,185.865,-63.956,-179.187,9.174,149.569
C00707=1122.850,185.651,-63.935,-179.188,9.172,149.569
C00708=1122.854,185.438,-63.914,-179.190,9.169,149.569
C00709=1122.857,185.223,-63.894,-179.193,9.166,149.569
C00710=1122.861,185.009,-63.873,-179.195,9.164,149.569
C00711=1122.865,184.795,-63.852,-179.197,9.162,149.569
C00712=1122.868,184.581,-63.832,-179.199,9.159,149.569
C00713=1122.873,184.367,-63.811,-179.201,9.156,149.569
C00714=1122.877,184.119,-63.787,-179.204,9.153,149.569
C00715=1122.882,183.870,-63.764,-179.207,9.150,149.569
C00716=1122.886,183.620,-63.739,-179.209,9.147,149.569
C00717=1122.891,183.372,-63.715,-179.212,9.144,149.569
C00718=1122.895,183.123,-63.691,-179.214,9.141,149.569
C00719=1122.900,182.875,-63.667,-179.217,9.138,149.569
C00720=1122.905,182.626,-63.644,-179.220,9.135,149.569
C00721=1122.909,182.377,-63.620,-179.222,9.132,149.569
C00722=1122.914,182.128,-63.597,-179.225,9.128,149.569
C00723=1122.918,181.880,-63.572,-179.228,9.125,149.569
C00724=1122.923,181.631,-63.549,-179.230,9.122,149.568
C00725=1122.927,181.382,-63.525,-179.233,9.119,149.569
C00726=1122.931,181.133,-63.501,-179.236,9.116,149.569
C00727=1122.936,180.883,-63.478,-179.239,9.112,149.569
C00728=1122.940,180.635,-63.454,-179.241,9.109,149.569
C00729=1122.945,180.386,-63.431,-179.244,9.106,149.568
C00730=1122.949,180.138,-63.406,-179.248,9.103,149.569
C00731=1122.954,179.889,-63.383,-179.250,9.099,149.569
C00732=1122.959,179.640,-63.360,-179.253,9.096,149.569
C00733=1122.963,179.391,-63.336,-179.256,9.092,149.568
C00734=1122.968,179.142,-63.312,-179.258,9.089,149.568
C00735=1122.973,178.893,-63.289,-179.260,9.087,149.568
C00736=1122.977,178.645,-63.265,-179.262,9.083,149.568
C00737=1122.982,178.396,-63.241,-179.265,9.080,149.568
C00738=1122.986,178.147,-63.218,-179.267,9.078,149.568
C00739=1122.991,177.898,-63.195,-179.269,9.075,149.568
C00740=1122.995,177.649,-63.171,-179.271,9.072,149.568
C00741=1123.000,177.400,-63.147,-179.273,9.069,149.568
C00742=1123.005,177.151,-63.124,-179.275,9.066,149.568
C00743=1123.010,176.902,-63.101,-179.277,9.063,149.568
C00744=1123.014,176.654,-63.077,-179.280,9.060,149.567
C00745=1123.018,176.405,-63.054,-179.282,9.057,149.567
C00746=1123.023,176.156,-63.030,-179.284,9.054,149.567
C00747=1123.027,175.907,-63.007,-179.286,9.051,149.567
C00748=1123.032,175.658,-62.984,-179.288,9.048,149.567
C00749=1123.037,175.409,-62.960,-179.290,9.045,149.567
C00750=1123.041,175.160,-62.936,-179.293,9.042,149.567
C00751=1123.046,174.911,-62.913,-179.295,9.039,149.567
C00752=1123.050,174.663,-62.890,-179.297,9.037,149.567
C00753=1123.054,174.414,-62.867,-179.299,9.033,149.567
C00754=1123.059,174.165,-62.843,-179.302,9.030,149.567
C00755=1123.064,173.916,-62.820,-179.303,9.028,149.566
C00756=1123.069,173.667,-62.797,-179.306,9.025,149.566
C00757=1123.074,173.418,-62.774,-179.308,9.021,149.566
C00758=1123.078,173.169,-62.751,-179.310,9.019,149.566
C00759=1123.083,172.920,-62.728,-179.312,9.016,149.566
C00760=1123.087,172.671,-62.704,-179.315,9.013,149.566
C00761=1123.092,172.422,-62.681,-179.317,9.009,149.566
C00762=1123.096,172.209,-62.661,-179.319,9.007,149.566
C00763=1123.099,171.995,-62.641,-179.321,9.004,149.566
C00764=1123.104,171.780,-62.621,-179.323,9.002,149.566
C00765=1123.107,171.566,-62.601,-179.325,8.999,149.566
C00766=1123.111,171.352,-62.581,-179.327,8.996,149.565
C00767=1123.115,171.138,-62.561,-179.328,8.994,149.565
C00768=1123.119,170.924,-62.542,-179.330,8.992,149.565
C00769=1123.123,170.711,-62.522,-179.333,8.988,149.565
C00770=1123.128,170.462,-62.499,-179.334,8.986,149.565
C00771=1123.132,170.212,-62.475,-179.337,8.983,149.565
C00772=1123.136,169.964,-62.452,-179.339,8.980,149.565
C00773=1123.141,169.714,-62.430,-179.341,8.976,149.565
C00774=1123.146,169.465,-62.406,-179.343,8.974,149.565
C00775=1123.151,169.217,-62.383,-179.346,8.971,149.565
C00776=1123.155,168.968,-62.361,-179.348,8.967,149.565
C00777=1123.160,168.719,-62.337,-179.350,8.964,149.564
C00778=1123.164,168.470,-62.315,-179.353,8.961,149.564
C00779=1123.169,168.221,-62.292,-179.355,8.958,149.564
C00780=1123.174,167.972,-62.269,-179.357,8.955,149.564
C00781=1123.178,167.724,-62.246,-179.359,8.952,149.564
C00782=1123.183,167.475,-62.223,-179.362,8.949,149.564
C00783=1123.188,167.225,-62.200,-179.365,8.946,149.564
C00784=1123.192,166.976,-62.177,-179.367,8.942,149.564
C00785=1123.197,166.728,-62.154,-179.369,8.939,149.564
C00786=1123.201,166.479,-62.132,-179.372,8.936,149.564
C00787=1123.206,166.229,-62.109,-179.374,8.933,149.563
C00788=1123.210,165.981,-62.086,-179.376,8.930,149.563
C00789=1123.216,165.732,-62.063,-179.378,8.927,149.563
C00790=1123.221,165.483,-62.041,-179.381,8.924,149.563
C00791=1123.224,165.234,-62.018,-179.383,8.921,149.563
C00792=1123.229,164.985,-61.995,-179.385,8.917,149.563
C00793=1123.234,164.736,-61.973,-179.388,8.914,149.563
C00794=1123.239,164.487,-61.949,-179.390,8.911,149.563
C00795=1123.243,164.239,-61.927,-179.392,8.908,149.563
C00796=1123.248,163.989,-61.904,-179.395,8.905,149.563
C00797=1123.252,163.741,-61.882,-179.397,8.901,149.562
C00798=1123.257,163.492,-61.860,-179.400,8.898,149.562
C00799=1123.261,163.243,-61.836,-179.402,8.895,149.562
C00800=1123.266,162.994,-61.815,-179.404,8.891,149.562
C00801=1123.271,162.745,-61.791,-179.407,8.888,149.562
C00802=1123.275,162.496,-61.769,-179.409,8.885,149.562
C00803=1123.280,162.247,-61.746,-179.411,8.882,149.562
C00804=1123.285,161.998,-61.724,-179.414,8.879,149.562
C00805=1123.289,161.749,-61.701,-179.416,8.876,149.562
C00806=1123.294,161.499,-61.679,-179.418,8.872,149.562
C00807=1123.298,161.251,-61.656,-179.421,8.869,149.561
C00808=1123.303,161.002,-61.634,-179.423,8.866,149.561
C00809=1123.307,160.753,-61.611,-179.426,8.862,149.561
C00810=1123.312,160.504,-61.589,-179.428,8.859,149.561
C00811=1123.317,160.255,-61.566,-179.431,8.856,149.561
C00812=1123.322,160.007,-61.544,-179.433,8.853,149.561
C00813=1123.326,159.757,-61.522,-179.435,8.850,149.561
C00814=1123.331,159.508,-61.499,-179.437,8.846,149.561
C00815=1123.335,159.260,-61.477,-179.440,8.843,149.561
C00816=1123.340,159.010,-61.455,-179.442,8.840,149.561
C00817=1123.344,158.761,-61.432,-179.444,8.836,149.560
C00818=1123.348,158.547,-61.413,-179.447,8.833,149.560
C00819=1123.353,158.333,-61.394,-179.448,8.831,149.560
C00820=1123.357,158.119,-61.374,-179.451,8.827,149.560
C00821=1123.361,157.905,-61.355,-179.453,8.824,149.560
C00822=1123.365,157.690,-61.336,-179.455,8.822,149.560
C00823=1123.369,157.476,-61.317,-179.457,8.818,149.560
C00824=1123.372,157.262,-61.299,-179.459,8.816,149.560
C00825=1123.376,157.048,-61.280,-179.461,8.813,149.560
C00826=1123.381,156.799,-61.257,-179.464,8.810,149.559
C00827=1123.386,156.551,-61.235,-179.466,8.806,149.559
C00828=1123.390,156.301,-61.213,-179.469,8.803,149.559
C00829=1123.395,156.053,-61.191,-179.471,8.799,149.559
C00830=1123.400,155.803,-61.168,-179.474,8.796,149.559
C00831=1123.404,155.554,-61.146,-179.476,8.792,149.559
C00832=1123.409,155.306,-61.124,-179.478,8.789,149.559
C00833=1123.413,155.056,-61.102,-179.480,8.786,149.558
C00834=1123.418,154.808,-61.080,-179.484,8.782,149.558
C00835=1123.422,154.558,-61.058,-179.486,8.778,149.558
C00836=1123.428,154.309,-61.036,-179.488,8.775,149.558
C00837=1123.432,154.060,-61.014,-179.490,8.772,149.558
C00838=1123.437,153.811,-60.992,-179.493,8.768,149.558
C00839=1123.441,153.562,-60.970,-179.496,8.764,149.558
C00840=1123.446,153.313,-60.948,-179.498,8.761,149.557
C00841=1123.451,153.065,-60.927,-179.501,8.757,149.557
C00842=1123.455,152.815,-60.904,-179.503,8.753,149.557
C00843=1123.460,152.567,-60.883,-179.505,8.750,149.557
C00844=1123.465,152.317,-60.860,-179.508,8.746,149.557
C00845=1123.470,152.068,-60.838,-179.511,8.743,149.557
C00846=1123.474,151.819,-60.816,-179.513,8.739,149.557
C00847=1123.479,151.570,-60.795,-179.515,8.735,149.556
C00848=1123.483,151.321,-60.773,-179.518,8.732,149.556
C00849=1123.488,151.072,-60.751,-179.520,8.728,149.556
C00850=1123.493,150.824,-60.729,-179.523,8.724,149.556
C00851=1123.497,150.574,-60.707,-179.525,8.721,149.556
C00852=1123.503,150.325,-60.686,-179.528,8.717,149.556
C00853=1123.507,150.076,-60.664,-179.530,8.713,149.555
C00854=1123.512,149.827,-60.643,-179.533,8.710,149.555
C00855=1123.517,149.579,-60.621,-179.535,8.706,149.555
C00856=1123.521,149.329,-60.599,-179.537,8.702,149.555
C00857=1123.526,149.081,-60.577,-179.540,8.698,149.555
C00858=1123.530,148.831,-60.556,-179.543,8.695,149.555
C00859=1123.535,148.582,-60.534,-179.545,8.691,149.554
C00860=1123.540,148.333,-60.512,-179.547,8.687,149.554
C00861=1123.544,148.084,-60.490,-179.550,8.683,149.554
C00862=1123.549,147.835,-60.470,-179.553,8.680,149.554
C00863=1123.554,147.586,-60.448,-179.555,8.676,149.554
C00864=1123.558,147.337,-60.426,-179.557,8.672,149.553
C00865=1123.563,147.088,-60.405,-179.560,8.668,149.553
C00866=1123.568,146.839,-60.384,-179.562,8.664,149.553
C00867=1123.572,146.590,-60.362,-179.565,8.661,149.553
C00868=1123.577,146.341,-60.340,-179.567,8.657,149.553
C00869=1123.582,146.092,-60.319,-179.570,8.653,149.552
C00870=1123.586,145.843,-60.298,-179.572,8.649,149.552
C00871=1123.591,145.594,-60.277,-179.575,8.645,149.552
C00872=1123.596,145.345,-60.255,-179.578,8.641,149.552
C00873=1123.601,145.096,-60.233,-179.580,8.637,149.551
C00874=1123.604,144.882,-60.215,-179.581,8.635,149.551
C00875=1123.609,144.667,-60.197,-179.582,8.632,149.551
C00876=1123.613,144.453,-60.178,-179.584,8.629,149.551
C00877=1123.616,144.238,-60.160,-179.585,8.626,149.550
C00878=1123.621,144.024,-60.141,-179.586,8.623,149.550
C00879=1123.625,143.810,-60.124,-179.588,8.620,149.550
C00880=1123.629,143.596,-60.105,-179.589,8.617,149.549
C00881=1123.633,143.382,-60.087,-179.590,8.615,149.549
C00882=1123.638,143.132,-60.066,-179.592,8.611,149.549
C00883=1123.642,142.883,-60.044,-179.593,8.608,149.548
C00884=1123.647,142.634,-60.023,-179.595,8.604,149.548
C00885=1123.651,142.386,-60.002,-179.596,8.601,149.548
C00886=1123.656,142.136,-59.981,-179.598,8.597,149.547
C00887=1123.661,141.887,-59.959,-179.600,8.594,149.547
C00888=1123.665,141.638,-59.938,-179.601,8.591,149.547
C00889=1123.670,141.389,-59.917,-179.603,8.587,149.546
C00890=1123.675,141.140,-59.896,-179.604,8.584,149.546
C00891=1123.680,140.891,-59.875,-179.606,8.581,149.546
C00892=1123.684,140.642,-59.853,-179.607,8.578,149.545
C00893=1123.689,140.393,-59.832,-179.609,8.574,149.545
C00894=1123.694,140.143,-59.811,-179.610,8.571,149.545
C00895=1123.698,139.895,-59.790,-179.612,8.568,149.544
C00896=1123.704,139.646,-59.769,-179.613,8.565,149.544
C00897=1123.707,139.396,-59.749,-179.615,8.561,149.544
C00898=1123.712,139.147,-59.727,-179.616,8.558,149.543
C00899=1123.717,138.898,-59.706,-179.618,8.555,149.543
C00900=1123.722,138.649,-59.686,-179.619,8.551,149.543
C00901=1123.727,138.401,-59.664,-179.621,8.548,149.542
C00902=1123.732,138.151,-59.643,-179.623,8.544,149.542
C00903=1123.736,137.902,-59.622,-179.625,8.541,149.542
C00904=1123.741,137.653,-59.600,-179.627,8.538,149.542
C00905=1123.745,137.404,-59.580,-179.628,8.535,149.541
C00906=1123.750,137.155,-59.559,-179.630,8.531,149.541
C00907=1123.755,136.906,-59.538,-179.631,8.528,149.540
C00908=1123.760,136.657,-59.517,-179.633,8.525,149.540
C00909=1123.765,136.408,-59.496,-179.634,8.521,149.540
C00910=1123.769,136.158,-59.475,-179.636,8.518,149.540
C00911=1123.774,135.909,-59.454,-179.638,8.515,149.539
C00912=1123.778,135.660,-59.434,-179.639,8.512,149.539
C00913=1123.783,135.411,-59.413,-179.641,8.508,149.539
C00914=1123.788,135.162,-59.392,-179.642,8.505,149.538
C00915=1123.793,134.913,-59.371,-179.644,8.501,149.538
C00916=1123.797,134.664,-59.351,-179.646,8.498,149.538
C00917=1123.802,134.415,-59.330,-179.647,8.495,149.537
C00918=1123.807,134.166,-59.309,-179.649,8.491,149.537
C00919=1123.812,133.917,-59.288,-179.651,8.489,149.537
C00920=1123.816,133.668,-59.268,-179.652,8.485,149.536
C00921=1123.821,133.418,-59.247,-179.654,8.481,149.536
C00922=1123.825,133.170,-59.226,-179.656,8.479,149.536
C00923=1123.830,132.920,-59.205,-179.657,8.475,149.536
C00924=1123.835,132.671,-59.184,-179.659,8.472,149.535
C00925=1123.840,132.422,-59.163,-179.661,8.469,149.535
C00926=1123.844,132.173,-59.143,-179.663,8.465,149.535
C00927=1123.849,131.924,-59.122,-179.664,8.462,149.534
C00928=1123.854,131.675,-59.102,-179.666,8.458,149.534
C00929=1123.858,131.426,-59.081,-179.668,8.456,149.534
C00930=1123.863,131.211,-59.063,-179.669,8.452,149.534
C00931=1123.867,130.997,-59.045,-179.671,8.449,149.533
C00932=1123.871,130.782,-59.028,-179.672,8.446,149.533
C00933=1123.875,130.568,-59.011,-179.674,8.444,149.533
C00934=1123.880,130.354,-58.993,-179.675,8.441,149.533
C00935=1123.883,130.139,-58.975,-179.676,8.438,149.532
C00936=1123.887,129.925,-58.957,-179.678,8.436,149.532
C00937=1123.891,129.711,-58.940,-179.679,8.433,149.532
C00938=1123.896,129.462,-58.919,-179.681,8.429,149.532
C00939=1123.901,129.213,-58.898,-179.683,8.425,149.531
C00940=1123.906,128.963,-58.878,-179.684,8.423,149.531
C00941=1123.911,128.714,-58.858,-179.687,8.419,149.531
C00942=1123.915,128.465,-58.837,-179.688,8.415,149.530
C00943=1123.920,128.216,-58.816,-179.690,8.413,149.530
C00944=1123.925,127.967,-58.796,-179.692,8.409,149.530
C00945=1123.929,127.718,-58.776,-179.694,8.406,149.530
C00946=1123.934,127.468,-58.755,-179.695,8.403,149.529
C00947=1123.939,127.219,-58.735,-179.697,8.399,149.529
C00948=1123.943,126.970,-58.715,-179.699,8.396,149.529
C00949=1123.948,126.721,-58.694,-179.700,8.393,149.529
C00950=1123.953,126.472,-58.673,-179.702,8.389,149.528
C00951=1123.958,126.223,-58.653,-179.704,8.386,149.528
C00952=1123.962,125.973,-58.633,-179.705,8.383,149.528
C00953=1123.967,125.725,-58.613,-179.708,8.379,149.528
C00954=1123.973,125.476,-58.592,-179.709,8.375,149.527
C00955=1123.977,125.227,-58.572,-179.711,8.373,149.527
C00956=1123.982,124.977,-58.552,-179.713,8.369,149.527
C00957=1123.986,124.728,-58.532,-179.715,8.366,149.526
C00958=1123.991,124.479,-58.511,-179.716,8.362,149.526
C00959=1123.996,124.229,-58.491,-179.718,8.359,149.526
C00960=1124.000,123.980,-58.471,-179.720,8.356,149.526
C00961=1124.005,123.732,-58.450,-179.722,8.352,149.525
C00962=1124.010,123.482,-58.431,-179.723,8.349,149.525
C00963=1124.014,123.233,-58.410,-179.725,8.346,149.525
C00964=1124.020,122.984,-58.390,-179.727,8.342,149.525
C00965=1124.025,122.735,-58.370,-179.729,8.339,149.524
C00966=1124.029,122.486,-58.350,-179.731,8.336,149.524
C00967=1124.034,122.236,-58.330,-179.733,8.332,149.524
C00968=1124.038,121.987,-58.310,-179.734,8.328,149.523
C00969=1124.043,121.738,-58.289,-179.736,8.325,149.523
C00970=1124.047,121.489,-58.270,-179.738,8.322,149.523
C00971=1124.052,121.241,-58.250,-179.740,8.319,149.523
C00972=1124.058,120.991,-58.229,-179.741,8.315,149.522
C00973=1124.062,120.742,-58.209,-179.744,8.311,149.522
C00974=1124.067,120.492,-58.189,-179.745,8.309,149.522
C00975=1124.072,120.243,-58.169,-179.747,8.305,149.522
C00976=1124.077,119.994,-58.150,-179.749,8.302,149.521
C00977=1124.081,119.746,-58.129,-179.751,8.298,149.521
C00978=1124.086,119.496,-58.110,-179.752,8.295,149.521
C00979=1124.091,119.247,-58.089,-179.754,8.292,149.521
C00980=1124.095,118.997,-58.070,-179.756,8.288,149.520
C00981=1124.100,118.749,-58.050,-179.758,8.285,149.520
C00982=1124.105,118.500,-58.030,-179.760,8.281,149.520
C00983=1124.110,118.250,-58.010,-179.761,8.278,149.519
C00984=1124.114,118.001,-57.990,-179.763,8.274,149.519
C00985=1124.119,117.752,-57.970,-179.766,8.271,149.519
C00986=1124.123,117.538,-57.953,-179.767,8.268,149.519
C00987=1124.127,117.323,-57.936,-179.769,8.265,149.519
C00988=1124.132,117.108,-57.919,-179.770,8.262,149.518
C00989=1124.136,116.894,-57.902,-179.772,8.259,149.518
C00990=1124.140,116.679,-57.885,-179.774,8.256,149.518
C00991=1124.144,116.465,-57.868,-179.775,8.253,149.517
C00992=1124.148,116.250,-57.850,-179.776,8.250,149.517
C00993=1124.152,116.036,-57.834,-179.778,8.247,149.517
C00994=1124.157,115.787,-57.815,-179.780,8.244,149.517
C00995=1124.161,115.537,-57.795,-179.782,8.240,149.517
C00996=1124.166,115.289,-57.775,-179.784,8.237,149.516
C00997=1124.171,115.039,-57.755,-179.786,8.233,149.516
C00998=1124.176,114.790,-57.736,-179.788,8.229,149.516
C00999=1124.180,114.541,-57.715,-179.790,8.226,149.515
C01000=1124.186,114.292,-57.696,-179.792,8.222,149.515
C01001=1124.191,114.042,-57.676,-179.793,8.220,149.515
C01002=1124.195,113.793,-57.657,-179.795,8.216,149.515
C01003=1124.201,113.544,-57.637,-179.797,8.212,149.514
C01004=1124.205,113.295,-57.617,-179.799,8.209,149.514
C01005=1124.209,113.046,-57.598,-179.801,8.205,149.514
C01006=1124.214,112.797,-57.579,-179.803,8.201,149.513
C01007=1124.219,112.547,-57.559,-179.805,8.198,149.513
C01008=1124.224,112.298,-57.539,-179.807,8.194,149.513
C01009=1124.229,112.049,-57.520,-179.809,8.191,149.513
C01010=1124.234,111.799,-57.500,-179.810,8.187,149.512
C01011=1124.238,111.551,-57.481,-179.812,8.184,149.512
C01012=1124.243,111.302,-57.461,-179.814,8.181,149.512
C01013=1124.248,111.052,-57.442,-179.816,8.177,149.512
C01014=1124.253,110.803,-57.422,-179.819,8.173,149.512
C01015=1124.258,110.554,-57.403,-179.821,8.170,149.511
C01016=1124.262,110.305,-57.384,-179.823,8.165,149.511
C01017=1124.267,110.056,-57.364,-179.826,8.162,149.511
C01018=1124.272,109.806,-57.345,-179.828,8.157,149.511
C01019=1124.277,109.557,-57.325,-179.830,8.154,149.510
C01020=1124.281,109.308,-57.306,-179.833,8.150,149.510
C01021=1124.286,109.058,-57.287,-179.835,8.146,149.510
C01022=1124.291,108.810,-57.267,-179.837,8.143,149.510
C01023=1124.296,108.560,-57.248,-179.840,8.138,149.510
C01024=1124.301,108.311,-57.229,-179.842,8.135,149.509
C01025=1124.305,108.062,-57.209,-179.845,8.131,149.509
C01026=1124.311,107.813,-57.190,-179.847,8.127,149.509
C01027=1124.315,107.563,-57.172,-179.849,8.122,149.508
C01028=1124.320,107.314,-57.152,-179.851,8.119,149.508
C01029=1124.325,107.065,-57.133,-179.854,8.115,149.508
C01030=1124.329,106.815,-57.114,-179.856,8.111,149.508
C01031=1124.335,106.567,-57.094,-179.858,8.108,149.508
C01032=1124.339,106.317,-57.075,-179.860,8.103,149.507
C01033=1124.344,106.068,-57.057,-179.862,8.100,149.507
C01034=1124.349,105.818,-57.037,-179.865,8.095,149.507
C01035=1124.354,105.570,-57.018,-179.867,8.092,149.506
C01036=1124.358,105.320,-56.999,-179.869,8.088,149.506
C01037=1124.363,105.072,-56.980,-179.871,8.084,149.506
C01038=1124.368,104.821,-56.961,-179.873,8.080,149.506
C01039=1124.373,104.572,-56.942,-179.876,8.076,149.505
C01040=1124.378,104.324,-56.923,-179.877,8.072,149.505
C01041=1124.383,104.074,-56.904,-179.879,8.068,149.505
C01042=1124.387,103.860,-56.888,-179.881,8.065,149.504
C01043=1124.391,103.645,-56.871,-179.883,8.061,149.504
C01044=1124.395,103.430,-56.855,-179.884,8.058,149.504
C01045=1124.399,103.215,-56.839,-179.887,8.055,149.504
C01046=1124.403,103.001,-56.823,-179.889,8.051,149.503
C01047=1124.408,102.787,-56.806,-179.890,8.047,149.503
C01048=1124.411,102.571,-56.790,-179.892,8.045,149.503
C01049=1124.416,102.357,-56.774,-179.894,8.041,149.503
C01050=1124.420,102.108,-56.755,-179.895,8.037,149.502
C01051=1124.426,101.858,-56.736,-179.898,8.033,149.502
C01052=1124.430,101.610,-56.717,-179.900,8.029,149.501
C01053=1124.435,101.361,-56.698,-179.902,8.026,149.501
C01054=1124.440,101.111,-56.680,-179.903,8.022,149.501
C01055=1124.445,100.862,-56.660,-179.906,8.017,149.501
C01056=1124.449,100.612,-56.642,-179.908,8.014,149.500
C01057=1124.454,100.364,-56.623,-179.910,8.010,149.500
C01058=1124.460,100.114,-56.605,-179.911,8.006,149.500
C01059=1124.464,99.865,-56.586,-179.913,8.001,149.499
C01060=1124.469,99.615,-56.567,-179.915,7.998,149.499
C01061=1124.474,99.367,-56.548,-179.917,7.994,149.498
C01062=1124.478,99.117,-56.530,-179.919,7.990,149.498
C01063=1124.484,98.867,-56.512,-179.921,7.986,149.498
C01064=1124.489,98.619,-56.493,-179.923,7.982,149.497
C01065=1124.493,98.369,-56.475,-179.925,7.978,149.497
C01066=1124.498,98.120,-56.455,-179.926,7.974,149.496
C01067=1124.503,97.871,-56.437,-179.928,7.971,149.496
C01068=1124.507,97.622,-56.418,-179.930,7.967,149.496
C01069=1124.513,97.372,-56.400,-179.932,7.962,149.495
C01070=1124.518,97.123,-56.382,-179.934,7.958,149.495
C01071=1124.522,96.874,-56.363,-179.935,7.954,149.495
C01072=1124.527,96.624,-56.344,-179.937,7.951,149.494
C01073=1124.532,96.375,-56.326,-179.939,7.947,149.494
C01074=1124.537,96.127,-56.307,-179.941,7.943,149.493
C01075=1124.541,95.877,-56.289,-179.942,7.939,149.493
C01076=1124.547,95.627,-56.270,-179.944,7.935,149.493
C01077=1124.552,95.378,-56.252,-179.946,7.931,149.492
C01078=1124.556,95.129,-56.233,-179.948,7.927,149.492
C01079=1124.561,94.880,-56.215,-179.950,7.923,149.492
C01080=1124.566,94.630,-56.197,-179.951,7.919,149.491
C01081=1124.571,94.381,-56.179,-179.953,7.916,149.491
C01082=1124.575,94.132,-56.160,-179.954,7.912,149.490
C01083=1124.580,93.883,-56.142,-179.956,7.908,149.490
C01084=1124.585,93.633,-56.124,-179.958,7.904,149.489
C01085=1124.591,93.384,-56.105,-179.959,7.900,149.489
C01086=1124.596,93.135,-56.087,-179.961,7.896,149.489
C01087=1124.600,92.885,-56.069,-179.962,7.892,149.488
C01088=1124.604,92.636,-56.050,-179.964,7.888,149.488
C01089=1124.609,92.387,-56.032,-179.966,7.884,149.487
C01090=1124.614,92.138,-56.014,-179.967,7.881,149.487
C01091=1124.619,91.888,-55.995,-179.969,7.877,149.486
C01092=1124.624,91.639,-55.977,-179.970,7.872,149.486
C01093=1124.629,91.389,-55.959,-179.972,7.868,149.485
C01094=1124.634,91.140,-55.941,-179.973,7.865,149.485
C01095=1124.639,90.891,-55.923,-179.975,7.861,149.484
C01096=1124.644,90.642,-55.905,-179.976,7.857,149.484
C01097=1124.648,90.392,-55.887,-179.978,7.853,149.484
C01098=1124.652,90.178,-55.871,-179.979,7.850,149.483
C01099=1124.657,89.963,-55.855,-179.980,7.846,149.483
C01100=1124.661,89.748,-55.840,-179.981,7.843,149.482
C01101=1124.665,89.533,-55.824,-179.983,7.840,149.482
C01102=1124.669,89.319,-55.809,-179.984,7.836,149.482
C01103=1124.673,89.104,-55.793,-179.985,7.833,149.481
C01104=1124.678,88.889,-55.778,-179.986,7.830,149.481
C01105=1124.682,88.674,-55.763,-179.988,7.826,149.480
C01106=1124.687,88.425,-55.745,-179.990,7.822,149.480
C01107=1124.692,88.176,-55.727,-179.991,7.819,149.480
C01108=1124.697,87.927,-55.708,-179.992,7.815,149.479
C01109=1124.702,87.677,-55.690,-179.993,7.811,149.478
C01110=1124.707,87.428,-55.672,-179.995,7.807,149.478
C01111=1124.712,87.179,-55.654,-179.996,7.803,149.478
C01112=1124.716,86.929,-55.636,-179.998,7.799,149.477
C01113=1124.721,86.680,-55.618,-179.999,7.796,149.477
C01114=1124.725,86.431,-55.600,180.000,7.792,149.476
C01115=1124.731,86.181,-55.583,179.999,7.787,149.475
C01116=1124.735,85.932,-55.565,179.997,7.784,149.475
C01117=1124.740,85.683,-55.547,179.996,7.780,149.475
C01118=1124.745,85.434,-55.529,179.995,7.776,149.474
C01119=1124.750,85.185,-55.511,179.993,7.772,149.474
C01120=1124.755,84.936,-55.493,179.992,7.768,149.473
C01121=1124.760,84.686,-55.476,179.991,7.765,149.472
C01122=1124.765,84.437,-55.458,179.990,7.761,149.472
C01123=1124.770,84.187,-55.440,179.988,7.757,149.472
C01124=1124.775,83.938,-55.422,179.987,7.753,149.471
C01125=1124.780,83.689,-55.404,179.986,7.750,149.471
C01126=1124.785,83.439,-55.387,179.985,7.745,149.470
C01127=1124.790,83.190,-55.369,179.983,7.742,149.469
C01128=1124.794,82.941,-55.352,179.982,7.738,149.469
C01129=1124.799,82.691,-55.334,179.981,7.734,149.468
C01130=1124.804,82.442,-55.316,179.980,7.730,149.468
C01131=1124.809,82.192,-55.298,179.979,7.727,149.467
C01132=1124.814,81.943,-55.280,179.978,7.723,149.467
C01133=1124.819,81.693,-55.263,179.977,7.719,149.466
C01134=1124.824,81.444,-55.245,179.975,7.715,149.466
C01135=1124.828,81.195,-55.227,179.974,7.711,149.465
C01136=1124.833,80.946,-55.210,179.973,7.708,149.465
C01137=1124.838,80.696,-55.192,179.972,7.704,149.464
C01138=1124.844,80.448,-55.174,179.971,7.701,149.464
C01139=1124.849,80.198,-55.157,179.970,7.696,149.463
C01140=1124.853,79.949,-55.140,179.969,7.692,149.463
C01141=1124.858,79.699,-55.123,179.968,7.689,149.462
C01142=1124.863,79.450,-55.105,179.966,7.685,149.462
C01143=1124.868,79.201,-55.087,179.966,7.682,149.461
C01144=1124.873,78.951,-55.069,179.964,7.678,149.460
C01145=1124.877,78.702,-55.052,179.964,7.674,149.460
C01146=1124.883,78.453,-55.035,179.962,7.670,149.459
C01147=1124.887,78.203,-55.017,179.962,7.667,149.459
C01148=1124.893,77.954,-54.999,179.960,7.663,149.458
C01149=1124.897,77.705,-54.982,179.960,7.659,149.458
C01150=1124.902,77.455,-54.965,179.959,7.656,149.457
C01151=1124.907,77.206,-54.947,179.958,7.652,149.457
C01152=1124.911,76.956,-54.930,179.957,7.648,149.456
C01153=1124.916,76.707,-54.912,179.956,7.645,149.456
C01154=1124.921,76.492,-54.897,179.955,7.641,149.455
C01155=1124.926,76.278,-54.882,179.953,7.638,149.455
C01156=1124.930,76.063,-54.867,179.952,7.634,149.454
C01157=1124.934,75.848,-54.852,179.951,7.631,149.454
C01158=1124.938,75.633,-54.838,179.949,7.627,149.453
C01159=1124.942,75.419,-54.822,179.949,7.624,149.453
C01160=1124.946,75.203,-54.808,179.947,7.620,149.453
C01161=1124.951,74.989,-54.793,179.946,7.617,149.452
C01162=1124.956,74.739,-54.775,179.944,7.613,149.452
C01163=1124.960,74.491,-54.758,179.943,7.609,149.451
C01164=1124.965,74.241,-54.741,179.942,7.605,149.451
C01165=1124.971,73.991,-54.723,179.940,7.601,149.450
C01166=1124.975,73.742,-54.706,179.939,7.597,149.450
C01167=1124.980,73.492,-54.689,179.937,7.594,149.449
C01168=1124.985,73.244,-54.672,179.936,7.589,149.449
C01169=1124.990,72.994,-54.654,179.934,7.585,149.448
C01170=1124.995,72.745,-54.637,179.933,7.581,149.448
C01171=1125.000,72.495,-54.620,179.931,7.578,149.447
C01172=1125.005,72.246,-54.603,179.930,7.573,149.447
C01173=1125.009,71.996,-54.586,179.928,7.569,149.446
C01174=1125.015,71.747,-54.569,179.927,7.565,149.446
C01175=1125.019,71.498,-54.552,179.925,7.562,149.445
C01176=1125.024,71.249,-54.534,179.925,7.558,149.445
C01177=1125.029,70.999,-54.518,179.923,7.554,149.444
C01178=1125.034,70.749,-54.500,179.922,7.550,149.444
C01179=1125.040,70.500,-54.483,179.920,7.546,149.444
C01180=1125.044,70.251,-54.466,179.919,7.542,149.443
C01181=1125.049,70.002,-54.449,179.917,7.538,149.442
C01182=1125.054,69.752,-54.432,179.916,7.534,149.442
C01183=1125.059,69.502,-54.415,179.915,7.530,149.441
C01184=1125.064,69.254,-54.399,179.913,7.526,149.441
C01185=1125.069,69.004,-54.381,179.912,7.522,149.441
C01186=1125.073,68.755,-54.364,179.910,7.518,149.440
C01187=1125.079,68.505,-54.347,179.909,7.514,149.439
C01188=1125.084,68.256,-54.330,179.907,7.510,149.439
C01189=1125.088,68.007,-54.314,179.906,7.506,149.439
C01190=1125.093,67.757,-54.296,179.905,7.502,149.438
C01191=1125.098,67.508,-54.280,179.903,7.498,149.438
C01192=1125.104,67.258,-54.263,179.901,7.494,149.437
C01193=1125.108,67.009,-54.246,179.900,7.490,149.436
C01194=1125.113,66.759,-54.229,179.899,7.486,149.436
C01195=1125.118,66.510,-54.213,179.897,7.482,149.436
C01196=1125.123,66.261,-54.196,179.896,7.478,149.435
C01197=1125.128,66.012,-54.178,179.895,7.474,149.435
C01198=1125.132,65.762,-54.161,179.894,7.471,149.434
C01199=1125.137,65.513,-54.145,179.892,7.467,149.434
C01200=1125.143,65.264,-54.128,179.891,7.462,149.433
C01201=1125.147,65.014,-54.111,179.889,7.458,149.433
C01202=1125.153,64.765,-54.095,179.888,7.455,149.432
C01203=1125.158,64.515,-54.078,179.887,7.450,149.432
C01204=1125.162,64.266,-54.062,179.885,7.446,149.431
C01205=1125.167,64.017,-54.045,179.884,7.442,149.431
C01206=1125.173,63.767,-54.028,179.882,7.438,149.430
C01207=1125.177,63.517,-54.011,179.881,7.434,149.430
C01208=1125.182,63.269,-53.995,179.879,7.430,149.429
C01209=1125.187,63.019,-53.978,179.878,7.426,149.429
C01210=1125.191,62.804,-53.964,179.877,7.423,149.428
C01211=1125.196,62.589,-53.949,179.876,7.419,149.428
C01212=1125.200,62.374,-53.935,179.875,7.416,149.427
C01213=1125.204,62.159,-53.921,179.873,7.412,149.427
C01214=1125.208,61.944,-53.907,179.872,7.409,149.426
C01215=1125.213,61.729,-53.892,179.871,7.406,149.426
C01216=1125.217,61.515,-53.879,179.870,7.402,149.426
C01217=1125.221,61.300,-53.863,179.869,7.399,149.425
C01218=1125.226,61.050,-53.847,179.867,7.395,149.425
C01219=1125.231,60.801,-53.831,179.866,7.391,149.424
C01220=1125.236,60.552,-53.814,179.865,7.387,149.424
C01221=1125.241,60.302,-53.797,179.863,7.382,149.423
C01222=1125.246,60.052,-53.781,179.862,7.378,149.423
C01223=1125.251,59.803,-53.765,179.860,7.375,149.422
C01224=1125.256,59.554,-53.748,179.859,7.370,149.421
C01225=1125.260,59.305,-53.732,179.858,7.366,149.421
C01226=1125.266,59.055,-53.716,179.857,7.362,149.420
C01227=1125.271,58.806,-53.699,179.855,7.358,149.420
C01228=1125.275,58.556,-53.682,179.853,7.354,149.420
C01229=1125.281,58.307,-53.667,179.852,7.350,149.419
C01230=1125.285,58.057,-53.650,179.851,7.346,149.418
C01231=1125.290,57.808,-53.634,179.850,7.342,149.418
C01232=1125.296,57.558,-53.617,179.849,7.339,149.417
C01233=1125.301,57.309,-53.601,179.847,7.335,149.417
C01234=1125.305,57.060,-53.584,179.846,7.330,149.416
C01235=1125.311,56.810,-53.569,179.845,7.326,149.416
C01236=1125.315,56.561,-53.552,179.843,7.322,149.415
C01237=1125.320,56.312,-53.536,179.842,7.318,149.415
C01238=1125.325,56.062,-53.520,179.841,7.314,149.414
C01239=1125.330,55.813,-53.503,179.839,7.310,149.414
C01240=1125.335,55.563,-53.487,179.838,7.306,149.413
C01241=1125.340,55.314,-53.471,179.837,7.302,149.413
C01242=1125.346,55.064,-53.455,179.835,7.298,149.412
C01243=1125.351,54.815,-53.438,179.834,7.294,149.412
C01244=1125.355,54.565,-53.422,179.832,7.290,149.411
C01245=1125.361,54.316,-53.406,179.831,7.285,149.411
C01246=1125.365,54.066,-53.390,179.830,7.281,149.410
C01247=1125.370,53.817,-53.374,179.829,7.277,149.409
C01248=1125.375,53.567,-53.358,179.827,7.273,149.409
C01249=1125.380,53.318,-53.341,179.826,7.269,149.408
C01250=1125.386,53.069,-53.326,179.824,7.265,149.408
C01251=1125.390,52.820,-53.309,179.823,7.261,149.407
C01252=1125.396,52.570,-53.294,179.822,7.257,149.407
C01253=1125.400,52.321,-53.277,179.821,7.253,149.406
C01254=1125.405,52.071,-53.261,179.819,7.249,149.406
C01255=1125.410,51.821,-53.245,179.818,7.244,149.405
C01256=1125.415,51.572,-53.229,179.817,7.241,149.405
C01257=1125.421,51.323,-53.213,179.816,7.237,149.404
C01258=1125.425,51.073,-53.197,179.814,7.233,149.404
C01259=1125.431,50.824,-53.181,179.813,7.229,149.403
C01260=1125.435,50.574,-53.165,179.812,7.225,149.403
C01261=1125.440,50.325,-53.150,179.811,7.220,149.402
C01262=1125.445,50.076,-53.134,179.809,7.217,149.402
C01263=1125.450,49.826,-53.118,179.808,7.212,149.401
C01264=1125.455,49.577,-53.102,179.807,7.208,149.400
C01265=1125.460,49.327,-53.086,179.805,7.204,149.400
C01266=1125.464,49.113,-53.072,179.804,7.200,149.399
C01267=1125.469,48.898,-53.059,179.803,7.197,149.399
C01268=1125.473,48.682,-53.044,179.802,7.193,149.398
C01269=1125.478,48.467,-53.031,179.801,7.190,149.398
C01270=1125.481,48.252,-53.017,179.800,7.186,149.397
C01271=1125.486,48.038,-53.004,179.798,7.183,149.397
C01272=1125.490,47.822,-52.990,179.798,7.179,149.397
C01273=1125.494,47.608,-52.977,179.796,7.175,149.396
C01274=1125.500,47.358,-52.962,179.796,7.172,149.396
C01275=1125.504,47.109,-52.945,179.794,7.168,149.395
C01276=1125.509,46.859,-52.929,179.793,7.164,149.394
C01277=1125.515,46.610,-52.914,179.792,7.159,149.394
C01278=1125.519,46.360,-52.898,179.791,7.155,149.393
C01279=1125.524,46.111,-52.883,179.789,7.151,149.393
C01280=1125.529,45.862,-52.867,179.788,7.147,149.392
C01281=1125.534,45.612,-52.851,179.787,7.143,149.391
C01282=1125.540,45.362,-52.835,179.785,7.139,149.391
C01283=1125.544,45.113,-52.820,179.784,7.134,149.390
C01284=1125.550,44.864,-52.804,179.783,7.130,149.390
C01285=1125.554,44.614,-52.789,179.782,7.126,149.389
C01286=1125.560,44.364,-52.773,179.781,7.122,149.389
C01287=1125.564,44.115,-52.758,179.779,7.118,149.388
C01288=1125.569,43.865,-52.742,179.778,7.114,149.388
C01289=1125.575,43.616,-52.726,179.777,7.109,149.387
C01290=1125.579,43.367,-52.711,179.775,7.105,149.387
C01291=1125.585,43.117,-52.696,179.774,7.101,149.386
C01292=1125.589,42.867,-52.680,179.773,7.097,149.385
C01293=1125.595,42.618,-52.664,179.772,7.093,149.385
C01294=1125.599,42.369,-52.649,179.771,7.089,149.384
C01295=1125.605,42.119,-52.634,179.770,7.084,149.384
C01296=1125.610,41.869,-52.618,179.768,7.080,149.383
C01297=1125.614,41.620,-52.603,179.767,7.076,149.382
C01298=1125.620,41.371,-52.587,179.766,7.072,149.382
C01299=1125.625,41.121,-52.572,179.765,7.067,149.381
C01300=1125.630,40.872,-52.557,179.763,7.063,149.381
C01301=1125.634,40.622,-52.541,179.762,7.059,149.380
C01302=1125.639,40.373,-52.526,179.761,7.055,149.379
C01303=1125.645,40.124,-52.510,179.760,7.051,149.379
C01304=1125.650,39.874,-52.494,179.758,7.047,149.378
C01305=1125.655,39.625,-52.479,179.757,7.042,149.378
C01306=1125.660,39.376,-52.464,179.756,7.038,149.377
C01307=1125.664,39.126,-52.449,179.755,7.034,149.377
C01308=1125.670,38.876,-52.434,179.754,7.030,149.376
C01309=1125.675,38.626,-52.418,179.753,7.025,149.375
C01310=1125.680,38.377,-52.403,179.752,7.021,149.375
C01311=1125.685,38.128,-52.387,179.751,7.017,149.374
C01312=1125.690,37.879,-52.372,179.749,7.013,149.374
C01313=1125.695,37.628,-52.357,179.748,7.009,149.373
C01314=1125.700,37.379,-52.342,179.747,7.004,149.372
C01315=1125.705,37.130,-52.327,179.746,7.000,149.372
C01316=1125.710,36.880,-52.311,179.745,6.996,149.371
C01317=1125.715,36.631,-52.296,179.743,6.992,149.371
C01318=1125.721,36.381,-52.281,179.742,6.987,149.370
C01319=1125.725,36.132,-52.266,179.741,6.983,149.369
C01320=1125.731,35.883,-52.251,179.740,6.979,149.369
C01321=1125.736,35.633,-52.236,179.739,6.975,149.368
C01322=1125.740,35.417,-52.223,179.737,6.971,149.368
C01323=1125.744,35.202,-52.210,179.737,6.967,149.367
C01324=1125.749,34.987,-52.197,179.736,6.964,149.366
C01325=1125.753,34.773,-52.185,179.735,6.960,149.366
C01326=1125.757,34.557,-52.171,179.734,6.957,149.365
C01327=1125.761,34.342,-52.158,179.732,6.953,149.365
C01328=1125.766,34.127,-52.145,179.732,6.949,149.364
C01329=1125.770,33.912,-52.132,179.731,6.945,149.364
C01330=1125.775,33.663,-52.117,179.729,6.941,149.363
C01331=1125.781,33.414,-52.102,179.728,6.937,149.363
C01332=1125.785,33.164,-52.087,179.727,6.932,149.362
C01333=1125.790,32.914,-52.072,179.726,6.928,149.361
C01334=1125.795,32.664,-52.057,179.725,6.924,149.361
C01335=1125.800,32.415,-52.042,179.724,6.919,149.360
C01336=1125.805,32.166,-52.027,179.723,6.915,149.359
C01337=1125.810,31.916,-52.012,179.722,6.911,149.359
C01338=1125.815,31.667,-51.997,179.721,6.906,149.358
C01339=1125.821,31.417,-51.982,179.720,6.902,149.357
C01340=1125.825,31.168,-51.967,179.719,6.898,149.357
C01341=1125.830,30.918,-51.953,179.717,6.894,149.356
C01342=1125.836,30.669,-51.938,179.716,6.889,149.356
C01343=1125.840,30.419,-51.923,179.715,6.885,149.355
C01344=1125.845,30.170,-51.908,179.714,6.881,149.354
C01345=1125.851,29.920,-51.893,179.713,6.877,149.354
C01346=1125.855,29.671,-51.878,179.712,6.872,149.353
C01347=1125.860,29.421,-51.864,179.711,6.868,149.352
C01348=1125.866,29.172,-51.849,179.710,6.864,149.352
C01349=1125.871,28.922,-51.834,179.709,6.859,149.351
C01350=1125.876,28.672,-51.820,179.707,6.854,149.351
C01351=1125.881,28.423,-51.804,179.706,6.850,149.350
C01352=1125.886,28.173,-51.790,179.705,6.846,149.349
C01353=1125.891,27.925,-51.776,179.704,6.841,149.349
C01354=1125.896,27.675,-51.761,179.703,6.836,149.348
C01355=1125.902,27.425,-51.746,179.702,6.832,149.347
C01356=1125.907,27.176,-51.731,179.701,6.828,149.346
C01357=1125.912,26.926,-51.717,179.700,6.824,149.346
C01358=1125.917,26.676,-51.703,179.699,6.819,149.345
C01359=1125.921,26.427,-51.688,179.698,6.815,149.344
C01360=1125.927,26.177,-51.673,179.697,6.811,149.344
C01361=1125.932,25.928,-51.659,179.696,6.806,149.343
C01362=1125.936,25.679,-51.644,179.695,6.802,149.343
C01363=1125.941,25.429,-51.629,179.694,6.798,149.342
C01364=1125.946,25.179,-51.615,179.693,6.793,149.341
C01365=1125.953,24.930,-51.601,179.692,6.789,149.341
C01366=1125.957,24.681,-51.586,179.691,6.784,149.340
C01367=1125.962,24.431,-51.571,179.690,6.779,149.339
C01368=1125.967,24.181,-51.557,179.689,6.775,149.338
C01369=1125.972,23.932,-51.543,179.687,6.771,149.338
C01370=1125.977,23.682,-51.529,179.686,6.766,149.337
C01371=1125.982,23.433,-51.514,179.685,6.762,149.336
C01372=1125.987,23.183,-51.499,179.684,6.758,149.336
C01373=1125.993,22.934,-51.485,179.684,6.753,149.335
C01374=1125.998,22.684,-51.471,179.683,6.749,149.334
C01375=1126.003,22.434,-51.456,179.682,6.744,149.334
C01376=1126.008,22.185,-51.441,179.681,6.740,149.333
C01377=1126.013,21.936,-51.427,179.679,6.735,149.332
C01378=1126.017,21.720,-51.415,179.679,6.731,149.332
C01379=1126.021,21.505,-51.402,179.678,6.727,149.331
C01380=1126.026,21.290,-51.390,179.677,6.723,149.330
C01381=1126.030,21.075,-51.378,179.676,6.719,149.330
C01382=1126.035,20.860,-51.365,179.675,6.716,149.329
C01383=1126.039,20.644,-51.354,179.674,6.712,149.329
C01384=1126.044,20.429,-51.341,179.674,6.708,149.328
C01385=1126.048,20.214,-51.329,179.673,6.704,149.327
C01386=1126.053,19.964,-51.315,179.672,6.699,149.327
C01387=1126.058,19.715,-51.300,179.671,6.695,149.326
C01388=1126.063,19.465,-51.286,179.670,6.690,149.325
C01389=1126.068,19.216,-51.272,179.669,6.686,149.325
C01390=1126.073,18.966,-51.258,179.668,6.682,149.324
C01391=1126.078,18.716,-51.244,179.667,6.677,149.323
C01392=1126.083,18.467,-51.229,179.666,6.672,149.322
C01393=1126.089,18.218,-51.216,179.665,6.668,149.322
C01394=1126.094,17.968,-51.201,179.664,6.663,149.321
C01395=1126.099,17.718,-51.187,179.663,6.659,149.320
C01396=1126.104,17.469,-51.173,179.662,6.654,149.320
C01397=1126.109,17.220,-51.159,179.661,6.650,149.319
C01398=1126.114,16.970,-51.144,179.660,6.645,149.318
C01399=1126.119,16.720,-51.130,179.659,6.641,149.317
C01400=1126.125,16.471,-51.116,179.658,6.635,149.316
C01401=1126.130,16.221,-51.102,179.657,6.631,149.316
C01402=1126.135,15.972,-51.088,179.656,6.627,149.315
C01403=1126.140,15.722,-51.073,179.656,6.622,149.314
C01404=1126.145,15.473,-51.061,179.654,6.618,149.314
C01405=1126.150,15.223,-51.047,179.654,6.613,149.313
C01406=1126.155,14.973,-51.032,179.653,6.609,149.312
C01407=1126.160,14.724,-51.018,179.652,6.603,149.311
C01408=1126.165,14.475,-51.004,179.651,6.599,149.311
C01409=1126.170,14.225,-50.990,179.650,6.595,149.310
C01410=1126.176,13.975,-50.977,179.649,6.590,149.309
C01411=1126.180,13.726,-50.963,179.648,6.586,149.308
C01412=1126.185,13.476,-50.949,179.648,6.581,149.308
C01413=1126.191,13.227,-50.935,179.646,6.576,149.307
C01414=1126.196,12.977,-50.921,179.645,6.571,149.306
C01415=1126.201,12.727,-50.907,179.644,6.567,149.305
C01416=1126.206,12.478,-50.893,179.644,6.562,149.304
C01417=1126.211,12.229,-50.879,179.643,6.558,149.304
C01418=1126.216,11.978,-50.866,179.642,6.553,149.303
C01419=1126.221,11.729,-50.852,179.641,6.548,149.302
C01420=1126.226,11.480,-50.838,179.640,6.543,149.301
C01421=1126.232,11.230,-50.825,179.639,6.539,149.301
C01422=1126.236,10.981,-50.811,179.638,6.534,149.300
C01423=1126.241,10.731,-50.796,179.638,6.529,149.299
C01424=1126.247,10.481,-50.783,179.636,6.524,149.298
C01425=1126.252,10.232,-50.770,179.636,6.519,149.297
C01426=1126.256,9.982,-50.755,179.635,6.515,149.297
C01427=1126.262,9.733,-50.742,179.634,6.510,149.296
C01428=1126.267,9.483,-50.728,179.634,6.506,149.295
C01429=1126.272,9.234,-50.714,179.632,6.501,149.294
C01430=1126.277,8.984,-50.701,179.631,6.496,149.294
C01431=1126.283,8.735,-50.687,179.631,6.491,149.293
C01432=1126.287,8.485,-50.674,179.630,6.487,149.292
C01433=1126.293,8.236,-50.660,179.629,6.482,149.291
C01434=1126.297,8.020,-50.648,179.628,6.478,149.291
C01435=1126.302,7.805,-50.636,179.628,6.474,149.290
C01436=1126.306,7.590,-50.625,179.628,6.470,149.289
C01437=1126.310,7.374,-50.613,179.627,6.467,149.288
C01438=1126.315,7.159,-50.601,179.627,6.462,149.287
C01439=1126.319,6.943,-50.590,179.626,6.459,149.287
C01440=1126.323,6.728,-50.578,179.627,6.455,149.286
C01441=1126.329,6.513,-50.567,179.626,6.451,149.285
C01442=1126.333,6.264,-50.553,179.626,6.446,149.284
C01443=1126.339,6.014,-50.540,179.625,6.442,149.283
C01444=1126.344,5.764,-50.525,179.625,6.437,149.283
C01445=1126.349,5.515,-50.513,179.625,6.433,149.282
C01446=1126.354,5.265,-50.499,179.624,6.429,149.281
C01447=1126.359,5.016,-50.486,179.623,6.424,149.280
C01448=1126.364,4.766,-50.472,179.623,6.419,149.279
C01449=1126.370,4.517,-50.458,179.623,6.415,149.278
C01450=1126.374,4.267,-50.446,179.622,6.411,149.278
C01451=1126.380,4.018,-50.432,179.622,6.406,149.277
C01452=1126.384,3.768,-50.419,179.621,6.401,149.276
C01453=1126.390,3.518,-50.405,179.620,6.397,149.275
C01454=1126.394,3.269,-50.392,179.620,6.393,149.274
C01455=1126.400,3.019,-50.379,179.620,6.388,149.273
C01456=1126.405,2.770,-50.365,179.619,6.383,149.272
C01457=1126.410,2.520,-50.352,179.618,6.379,149.272
C01458=1126.415,2.270,-50.339,179.618,6.374,149.271
C01459=1126.421,2.021,-50.325,179.618,6.370,149.270
C01460=1126.426,1.771,-50.311,179.617,6.366,149.269
C01461=1126.431,1.521,-50.299,179.616,6.361,149.268
C01462=1126.436,1.272,-50.284,179.616,6.356,149.267
C01463=1126.441,1.022,-50.272,179.615,6.352,149.267
C01464=1126.447,0.773,-50.259,179.615,6.348,149.266
C01465=1126.451,0.523,-50.246,179.614,6.343,149.265
C01466=1126.456,0.274,-50.232,179.614,6.339,149.264
C01467=1126.461,0.024,-50.219,179.613,6.334,149.263
C01468=1126.467,-0.226,-50.206,179.612,6.329,149.263
C01469=1126.472,-0.475,-50.193,179.612,6.325,149.262
C01470=1126.477,-0.725,-50.179,179.612,6.321,149.261
C01471=1126.482,-0.974,-50.166,179.611,6.316,149.260
C01472=1126.487,-1.224,-50.153,179.610,6.312,149.259
C01473=1126.493,-1.474,-50.140,179.610,6.307,149.258
C01474=1126.498,-1.723,-50.127,179.609,6.302,149.257
C01475=1126.503,-1.973,-50.113,179.608,6.298,149.257
C01476=1126.508,-2.222,-50.100,179.608,6.293,149.256
C01477=1126.513,-2.472,-50.087,179.608,6.289,149.255
C01478=1126.518,-2.722,-50.074,179.607,6.285,149.254
C01479=1126.524,-2.971,-50.062,179.606,6.280,149.254
C01480=1126.529,-3.222,-50.048,179.606,6.276,149.253
C01481=1126.534,-3.470,-50.035,179.605,6.271,149.252
C01482=1126.539,-3.720,-50.022,179.604,6.266,149.251
C01483=1126.544,-3.970,-50.009,179.604,6.262,149.250
C01484=1126.549,-4.219,-49.996,179.603,6.257,149.249
C01485=1126.554,-4.469,-49.983,179.602,6.253,149.249
C01486=1126.560,-4.719,-49.970,179.602,6.249,149.248
C01487=1126.565,-4.968,-49.957,179.602,6.244,149.247
C01488=1126.570,-5.218,-49.945,179.601,6.239,149.246
C01489=1126.575,-5.468,-49.931,179.600,6.235,149.245
C01490=1126.580,-5.683,-49.920,179.599,6.231,149.245
C01491=1126.584,-5.898,-49.909,179.599,6.227,149.244
C01492=1126.588,-6.113,-49.898,179.599,6.223,149.243
C01493=1126.593,-6.329,-49.887,179.598,6.219,149.242
C01494=1126.597,-6.544,-49.875,179.598,6.215,149.242
C01495=1126.601,-6.760,-49.864,179.597,6.211,149.241
C01496=1126.607,-6.975,-49.854,179.596,6.207,149.240
C01497=1126.611,-7.190,-49.842,179.596,6.203,149.240
C01498=1126.616,-7.439,-49.830,179.595,6.199,149.239
C01499=1126.621,-7.690,-49.816,179.595,6.194,149.238
C01500=1126.626,-7.939,-49.803,179.594,6.190,149.237
C01501=1126.631,-8.188,-49.791,179.593,6.185,149.237
C01502=1126.636,-8.438,-49.778,179.593,6.181,149.236
C01503=1126.642,-8.688,-49.765,179.592,6.176,149.235
C01504=1126.647,-8.937,-49.752,179.591,6.171,149.234
C01505=1126.652,-9.187,-49.740,179.591,6.167,149.233
C01506=1126.657,-9.437,-49.727,179.590,6.162,149.233
C01507=1126.662,-9.687,-49.715,179.589,6.158,149.232
C01508=1126.668,-9.936,-49.701,179.589,6.153,149.231
C01509=1126.673,-10.186,-49.689,179.588,6.149,149.230
C01510=1126.677,-10.436,-49.676,179.587,6.144,149.229
C01511=1126.683,-10.685,-49.663,179.587,6.139,149.228
C01512=1126.688,-10.934,-49.651,179.586,6.135,149.228
C01513=1126.693,-11.184,-49.639,179.585,6.130,149.227
C01514=1126.699,-11.434,-49.626,179.585,6.125,149.226
C01515=1126.704,-11.684,-49.613,179.584,6.121,149.225
C01516=1126.709,-11.933,-49.600,179.583,6.116,149.224
C01517=1126.714,-12.183,-49.587,179.583,6.112,149.223
C01518=1126.719,-12.432,-49.575,179.582,6.107,149.223
C01519=1126.724,-12.682,-49.563,179.581,6.102,149.222
C01520=1126.729,-12.932,-49.550,179.581,6.098,149.221
C01521=1126.735,-13.181,-49.537,179.579,6.093,149.220
C01522=1126.740,-13.431,-49.525,179.579,6.088,149.219
C01523=1126.745,-13.681,-49.512,179.578,6.083,149.219
C01524=1126.750,-13.930,-49.500,179.577,6.079,149.218
C01525=1126.755,-14.179,-49.487,179.577,6.074,149.217
C01526=1126.760,-14.430,-49.475,179.576,6.069,149.216
C01527=1126.765,-14.679,-49.462,179.575,6.065,149.215
C01528=1126.771,-14.929,-49.450,179.575,6.060,149.215
C01529=1126.776,-15.179,-49.438,179.574,6.055,149.214
C01530=1126.781,-15.428,-49.425,179.573,6.051,149.213
C01531=1126.786,-15.677,-49.413,179.572,6.046,149.212
C01532=1126.792,-15.927,-49.401,179.572,6.041,149.211
C01533=1126.796,-16.177,-49.388,179.571,6.037,149.211
C01534=1126.801,-16.426,-49.375,179.570,6.032,149.210
C01535=1126.807,-16.676,-49.363,179.570,6.027,149.209
C01536=1126.812,-16.926,-49.351,179.569,6.023,149.208
C01537=1126.817,-17.176,-49.339,179.568,6.018,149.207
C01538=1126.822,-17.425,-49.326,179.567,6.012,149.206
C01539=1126.828,-17.675,-49.314,179.566,6.008,149.206
C01540=1126.833,-17.924,-49.302,179.566,6.003,149.205
C01541=1126.838,-18.173,-49.289,179.565,5.999,149.204
C01542=1126.844,-18.423,-49.277,179.564,5.994,149.203
C01543=1126.849,-18.673,-49.265,179.563,5.989,149.202
C01544=1126.854,-18.923,-49.253,179.563,5.984,149.202
C01545=1126.859,-19.173,-49.240,179.562,5.979,149.201
C01546=1126.864,-19.388,-49.229,179.561,5.975,149.200
C01547=1126.867,-19.603,-49.219,179.561,5.971,149.199
C01548=1126.873,-19.819,-49.208,179.560,5.967,149.199
C01549=1126.877,-20.035,-49.197,179.559,5.963,149.198
C01550=1126.882,-20.250,-49.188,179.559,5.959,149.197
C01551=1126.886,-20.466,-49.177,179.558,5.954,149.196
C01552=1126.890,-20.681,-49.167,179.557,5.950,149.196
C01553=1126.895,-20.897,-49.156,179.557,5.946,149.195
C01554=1126.900,-21.146,-49.143,179.556,5.942,149.194
C01555=1126.905,-21.396,-49.131,179.555,5.936,149.193
C01556=1126.911,-21.645,-49.119,179.554,5.932,149.193
C01557=1126.916,-21.895,-49.107,179.554,5.927,149.192
C01558=1126.921,-22.145,-49.096,179.553,5.922,149.191
C01559=1126.926,-22.394,-49.083,179.552,5.917,149.190
C01560=1126.931,-22.644,-49.071,179.551,5.913,149.189
C01561=1126.937,-22.894,-49.059,179.550,5.907,149.188
C01562=1126.942,-23.143,-49.047,179.550,5.902,149.188
C01563=1126.948,-23.393,-49.035,179.549,5.898,149.187
C01564=1126.953,-23.642,-49.024,179.548,5.892,149.186
C01565=1126.958,-23.891,-49.011,179.547,5.888,149.185
C01566=1126.963,-24.141,-48.999,179.547,5.883,149.184
C01567=1126.969,-24.391,-48.987,179.546,5.877,149.183
C01568=1126.974,-24.641,-48.976,179.545,5.873,149.182
C01569=1126.978,-24.890,-48.964,179.545,5.868,149.182
C01570=1126.984,-25.140,-48.952,179.543,5.863,149.181
C01571=1126.989,-25.390,-48.940,179.543,5.858,149.180
C01572=1126.995,-25.640,-48.928,179.542,5.852,149.179
C01573=1126.999,-25.889,-48.916,179.541,5.848,149.178
C01574=1127.004,-26.139,-48.904,179.541,5.844,149.177
C01575=1127.010,-26.389,-48.892,179.542,5.839,149.176
C01576=1127.015,-26.639,-48.880,179.544,5.835,149.175
C01577=1127.020,-26.888,-48.868,179.545,5.832,149.174
C01578=1127.026,-27.137,-48.857,179.545,5.828,149.173
C01579=1127.031,-27.387,-48.845,179.547,5.824,149.171
C01580=1127.036,-27.637,-48.834,179.547,5.820,149.170
C01581=1127.041,-27.887,-48.822,179.548,5.816,149.169
C01582=1127.046,-28.136,-48.809,179.549,5.812,149.168
C01583=1127.052,-28.386,-48.797,179.549,5.808,149.167
C01584=1127.057,-28.636,-48.786,179.550,5.804,149.166
C01585=1127.062,-28.886,-48.774,179.551,5.800,149.165
C01586=1127.067,-29.135,-48.762,179.551,5.796,149.164
C01587=1127.072,-29.385,-48.751,179.552,5.792,149.163
C01588=1127.078,-29.634,-48.739,179.552,5.788,149.162
C01589=1127.083,-29.884,-48.727,179.553,5.783,149.161
C01590=1127.088,-30.133,-48.715,179.553,5.780,149.160
C01591=1127.093,-30.383,-48.704,179.553,5.775,149.159
C01592=1127.099,-30.633,-48.692,179.554,5.771,149.158
C01593=1127.103,-30.883,-48.680,179.554,5.767,149.157
C01594=1127.109,-31.133,-48.668,179.554,5.763,149.156
C01595=1127.114,-31.383,-48.657,179.554,5.758,149.155
C01596=1127.120,-31.632,-48.646,179.554,5.754,149.154
C01597=1127.125,-31.881,-48.633,179.554,5.750,149.153
C01598=1127.130,-32.131,-48.621,179.554,5.746,149.152
C01599=1127.135,-32.380,-48.610,179.554,5.742,149.151
C01600=1127.140,-32.630,-48.598,179.553,5.737,149.150
C01601=1127.146,-32.880,-48.586,179.553,5.733,149.149
C01602=1127.150,-33.096,-48.577,179.553,5.729,149.149
C01603=1127.155,-33.311,-48.567,179.553,5.725,149.148
C01604=1127.159,-33.527,-48.556,179.552,5.721,149.147
C01605=1127.164,-33.742,-48.547,179.552,5.718,149.147
C01606=1127.168,-33.958,-48.536,179.552,5.714,149.146
C01607=1127.173,-34.173,-48.526,179.552,5.710,149.145
C01608=1127.177,-34.388,-48.516,179.551,5.706,149.144
C01609=1127.181,-34.604,-48.507,179.551,5.702,149.144
C01610=1127.187,-34.854,-48.495,179.550,5.697,149.143
C01611=1127.193,-35.104,-48.483,179.550,5.693,149.142
C01612=1127.198,-35.353,-48.472,179.549,5.688,149.141
C01613=1127.203,-35.603,-48.460,179.548,5.684,149.140
C01614=1127.208,-35.853,-48.449,179.547,5.678,149.140
C01615=1127.214,-36.102,-48.437,179.546,5.674,149.139
C01616=1127.218,-36.352,-48.426,179.546,5.669,149.138
C01617=1127.224,-36.602,-48.414,179.544,5.664,149.137
C01618=1127.228,-36.851,-48.403,179.543,5.659,149.136
C01619=1127.234,-37.101,-48.391,179.542,5.654,149.136
C01620=1127.239,-37.350,-48.380,179.541,5.649,149.135
C01621=1127.245,-37.601,-48.369,179.540,5.644,149.134
C01622=1127.250,-37.850,-48.358,179.539,5.640,149.133
C01623=1127.255,-38.100,-48.346,179.538,5.634,149.133
C01624=1127.260,-38.349,-48.335,179.537,5.629,149.132
C01625=1127.266,-38.599,-48.323,179.535,5.624,149.131
C01626=1127.270,-38.849,-48.312,179.534,5.619,149.130
C01627=1127.277,-39.099,-48.301,179.533,5.613,149.130
C01628=1127.281,-39.348,-48.289,179.531,5.608,149.129
C01629=1127.287,-39.598,-48.278,179.530,5.603,149.128
C01630=1127.292,-39.848,-48.266,179.528,5.597,149.128
C01631=1127.297,-40.097,-48.256,179.527,5.592,149.127
C01632=1127.303,-40.347,-48.244,179.525,5.587,149.126
C01633=1127.307,-40.597,-48.233,179.523,5.581,149.125
C01634=1127.313,-40.846,-48.221,179.522,5.576,149.125
C01635=1127.318,-41.096,-48.211,179.520,5.570,149.124
C01636=1127.323,-41.346,-48.200,179.518,5.565,149.123
C01637=1127.329,-41.595,-48.188,179.516,5.558,149.122
C01638=1127.334,-41.845,-48.177,179.515,5.553,149.122
C01639=1127.339,-42.094,-48.167,179.513,5.547,149.121
C01640=1127.345,-42.344,-48.155,179.511,5.541,149.120
C01641=1127.350,-42.595,-48.144,179.509,5.535,149.120
C01642=1127.355,-42.843,-48.133,179.507,5.530,149.119
C01643=1127.361,-43.094,-48.122,179.505,5.524,149.119
C01644=1127.366,-43.343,-48.111,179.504,5.518,149.117
C01645=1127.371,-43.593,-48.100,179.505,5.514,149.116
C01646=1127.376,-43.843,-48.089,179.505,5.509,149.115
C01647=1127.382,-44.093,-48.078,179.505,5.505,149.114
C01648=1127.387,-44.342,-48.067,179.505,5.499,149.113
C01649=1127.392,-44.591,-48.056,179.505,5.495,149.112
C01650=1127.397,-44.841,-48.046,179.506,5.490,149.111
C01651=1127.403,-45.091,-48.034,179.506,5.485,149.110
C01652=1127.408,-45.341,-48.023,179.506,5.481,149.109
C01653=1127.413,-45.591,-48.012,179.506,5.476,149.108
C01654=1127.418,-45.840,-48.002,179.506,5.471,149.107
C01655=1127.424,-46.091,-47.991,179.507,5.467,149.106
C01656=1127.429,-46.340,-47.980,179.506,5.462,149.105
C01657=1127.434,-46.590,-47.969,179.507,5.458,149.103
C01658=1127.439,-46.805,-47.960,179.507,5.454,149.103
C01659=1127.444,-47.021,-47.951,179.507,5.450,149.102
C01660=1127.448,-47.236,-47.941,179.507,5.445,149.101
C01661=1127.452,-47.453,-47.932,179.507,5.441,149.100
C01662=1127.457,-47.668,-47.922,179.508,5.437,149.099
C01663=1127.462,-47.884,-47.913,179.508,5.433,149.098
C01664=1127.466,-48.099,-47.904,179.508,5.429,149.097
C01665=1127.471,-48.315,-47.895,179.508,5.425,149.096
C01666=1127.476,-48.564,-47.883,179.508,5.420,149.095
C01667=1127.481,-48.814,-47.873,179.508,5.416,149.094
C01668=1127.487,-49.064,-47.862,179.508,5.410,149.093
C01669=1127.492,-49.313,-47.851,179.509,5.406,149.092
C01670=1127.497,-49.563,-47.840,179.509,5.401,149.091
C01671=1127.503,-49.812,-47.830,179.509,5.397,149.090
C01672=1127.508,-50.063,-47.819,179.509,5.392,149.088
C01673=1127.513,-50.312,-47.809,179.509,5.387,149.088
C01674=1127.518,-50.562,-47.797,179.510,5.383,149.086
C01675=1127.524,-50.811,-47.787,179.510,5.378,149.085
C01676=1127.529,-51.062,-47.776,179.510,5.373,149.084
C01677=1127.535,-51.311,-47.765,179.510,5.369,149.083
C01678=1127.540,-51.561,-47.755,179.511,5.364,149.082
C01679=1127.545,-51.811,-47.744,179.511,5.359,149.081
C01680=1127.550,-52.061,-47.734,179.511,5.355,149.080
C01681=1127.555,-52.310,-47.723,179.511,5.350,149.079
C01682=1127.561,-52.559,-47.713,179.511,5.345,149.078
C01683=1127.566,-52.810,-47.702,179.511,5.341,149.077
C01684=1127.571,-53.058,-47.691,179.511,5.336,149.076
C01685=1127.576,-53.309,-47.681,179.512,5.331,149.074
C01686=1127.582,-53.558,-47.670,179.512,5.327,149.074
C01687=1127.587,-53.808,-47.660,179.512,5.322,149.072
C01688=1127.592,-54.057,-47.649,179.512,5.317,149.071
C01689=1127.598,-54.308,-47.638,179.513,5.313,149.070
C01690=1127.604,-54.558,-47.628,179.513,5.308,149.069
C01691=1127.609,-54.807,-47.617,179.513,5.303,149.068
C01692=1127.614,-55.057,-47.607,179.514,5.299,149.067
C01693=1127.619,-55.306,-47.596,179.513,5.294,149.066
C01694=1127.624,-55.556,-47.585,179.514,5.289,149.065
C01695=1127.630,-55.806,-47.575,179.514,5.284,149.064
C01696=1127.635,-56.056,-47.564,179.514,5.280,149.063
C01697=1127.641,-56.306,-47.554,179.514,5.275,149.062
C01698=1127.646,-56.555,-47.543,179.515,5.271,149.060
C01699=1127.650,-56.805,-47.533,179.514,5.266,149.060
C01700=1127.656,-57.054,-47.523,179.515,5.262,149.058
C01701=1127.661,-57.304,-47.513,179.515,5.257,149.057
C01702=1127.666,-57.554,-47.502,179.515,5.252,149.056
C01703=1127.672,-57.804,-47.492,179.516,5.247,149.055
C01704=1127.677,-58.054,-47.482,179.516,5.242,149.054
C01705=1127.683,-58.303,-47.471,179.516,5.238,149.053
C01706=1127.687,-58.553,-47.460,179.516,5.233,149.052
C01707=1127.693,-58.802,-47.450,179.517,5.229,149.051
C01708=1127.698,-59.052,-47.440,179.516,5.224,149.050
C01709=1127.703,-59.302,-47.429,179.517,5.220,149.049
C01710=1127.709,-59.552,-47.419,179.517,5.215,149.048
C01711=1127.714,-59.802,-47.408,179.517,5.211,149.047
C01712=1127.720,-60.052,-47.398,179.517,5.205,149.046
C01713=1127.725,-60.301,-47.388,179.518,5.201,149.045
C01714=1127.731,-60.629,-47.374,179.516,5.194,149.043
C01715=1127.739,-60.958,-47.361,179.515,5.187,149.042
C01716=1127.746,-61.285,-47.347,179.514,5.180,149.041
C01717=1127.752,-61.614,-47.333,179.512,5.173,149.040
C01718=1127.758,-61.863,-47.323,179.511,5.167,149.039
C01719=1127.763,-62.113,-47.313,179.511,5.163,149.038
C01720=1127.769,-62.362,-47.303,179.510,5.157,149.037
C01721=1127.774,-62.613,-47.293,179.509,5.151,149.036
C01722=1127.779,-62.863,-47.283,179.508,5.146,149.036
C01723=1127.785,-63.112,-47.273,179.507,5.141,149.035
C01724=1127.790,-63.362,-47.262,179.506,5.135,149.034
C01725=1127.795,-63.612,-47.253,179.505,5.130,149.033
C01726=1127.800,-63.861,-47.243,179.504,5.124,149.032
C01727=1127.806,-64.111,-47.232,179.504,5.120,149.031
C01728=1127.811,-64.361,-47.222,179.503,5.114,149.030
C01729=1127.817,-64.610,-47.212,179.502,5.108,149.029
C01730=1127.839,-65.621,-47.173,178.902,6.226,149.449
C01731=1127.844,-65.871,-47.163,178.899,6.225,149.450
C01732=1127.849,-66.120,-47.152,178.897,6.224,149.450
C01733=1127.854,-66.370,-47.143,178.895,6.224,149.451
C01734=1127.859,-66.620,-47.132,178.892,6.223,149.451
C01735=1127.865,-66.869,-47.122,178.891,6.223,149.452
C01736=1127.870,-67.119,-47.112,178.889,6.222,149.452
C01737=1127.875,-67.369,-47.101,178.886,6.221,149.453
C01738=1127.881,-67.619,-47.091,178.884,6.221,149.453
C01739=1127.886,-67.868,-47.081,178.882,6.220,149.454
C01740=1127.891,-68.118,-47.071,178.879,6.220,149.454
C01741=1127.896,-68.368,-47.061,178.878,6.220,149.455
C01742=1127.902,-68.617,-47.050,178.876,6.219,149.455
C01743=1127.908,-68.867,-47.041,178.873,6.218,149.456
C01744=1127.913,-69.118,-47.030,178.871,6.217,149.456
C01745=1127.918,-69.367,-47.021,178.869,6.217,149.457
C01746=1127.923,-69.616,-47.010,178.866,6.216,149.458
C01747=1127.928,-69.867,-47.000,178.865,6.216,149.458
C01748=1127.934,-70.116,-46.990,178.863,6.215,149.458
C01749=1127.939,-70.366,-46.979,178.860,6.215,149.459
C01750=1127.944,-70.615,-46.970,178.858,6.214,149.459
C01751=1127.950,-70.866,-46.960,178.856,6.213,149.460
C01752=1127.955,-71.115,-46.950,178.854,6.214,149.461
C01753=1127.961,-71.365,-46.940,178.852,6.213,149.461
C01754=1127.966,-71.614,-46.930,178.850,6.212,149.462
C01755=1127.971,-71.864,-46.920,178.847,6.211,149.462
C01756=1127.976,-72.114,-46.909,178.845,6.211,149.463
C01757=1127.982,-72.364,-46.900,178.843,6.210,149.463
C01758=1127.987,-72.613,-46.890,178.841,6.210,149.464
C01759=1127.993,-72.863,-46.880,178.839,6.210,149.464
C01760=1127.998,-73.113,-46.869,178.836,6.209,149.465
C01761=1128.002,-73.362,-46.860,178.834,6.208,149.465
C01762=1128.008,-73.613,-46.850,178.832,6.207,149.466
C01763=1128.014,-73.862,-46.840,178.831,6.207,149.466
C01764=1128.020,-74.112,-46.830,178.828,6.207,149.467
C01765=1128.024,-74.362,-46.820,178.826,6.206,149.467
C01766=1128.030,-74.612,-46.810,178.824,6.205,149.468
C01767=1128.035,-74.861,-46.800,178.821,6.205,149.468
C01768=1128.040,-75.111,-46.790,178.820,6.205,149.469
C01769=1128.046,-75.360,-46.780,178.817,6.204,149.469
C01770=1128.051,-75.611,-46.770,178.815,6.203,149.470
C01771=1128.056,-75.860,-46.761,178.813,6.202,149.470
C01772=1128.061,-76.110,-46.751,178.811,6.202,149.471
C01773=1128.067,-76.360,-46.741,178.809,6.202,149.471
C01774=1128.072,-76.609,-46.731,178.807,6.201,149.472
C01775=1128.078,-76.881,-46.721,178.804,6.201,149.472
C01776=1128.084,-77.153,-46.710,178.802,6.200,149.473
C01777=1128.091,-77.424,-46.699,178.800,6.199,149.473
C01778=1128.096,-77.695,-46.688,178.797,6.199,149.474
C01779=1128.102,-77.946,-46.679,178.795,6.198,149.475
C01780=1128.106,-78.195,-46.669,178.794,6.198,149.475
C01781=1128.111,-78.445,-46.659,178.791,6.197,149.476
C01782=1128.117,-78.695,-46.650,178.789,6.196,149.476
C01783=1128.122,-78.944,-46.640,178.787,6.196,149.477
C01784=1128.128,-79.194,-46.629,178.785,6.195,149.477
C01785=1128.133,-79.444,-46.620,178.783,6.195,149.477
C01786=1128.139,-79.693,-46.610,178.781,6.194,149.478
C01787=1128.144,-79.943,-46.601,178.779,6.194,149.478
C01788=1128.149,-80.193,-46.591,178.776,6.193,149.479
C01789=1128.154,-80.443,-46.581,178.775,6.193,149.480
C01790=1128.160,-80.693,-46.572,178.772,6.192,149.480
C01791=1128.165,-80.942,-46.561,178.770,6.192,149.481
C01792=1128.170,-81.192,-46.553,178.768,6.191,149.481
C01793=1128.176,-81.442,-46.542,178.766,6.191,149.482
C01794=1128.181,-81.692,-46.533,178.764,6.190,149.482
C01795=1128.187,-81.941,-46.523,178.762,6.189,149.483
C01796=1128.192,-82.191,-46.514,178.760,6.189,149.483
C01797=1128.197,-82.441,-46.504,178.758,6.189,149.484
C01798=1128.202,-82.691,-46.495,178.755,6.188,149.484
C01799=1128.208,-82.941,-46.485,178.753,6.188,149.485
C01800=1128.213,-83.191,-46.476,178.751,6.187,149.485
C01801=1128.218,-83.440,-46.466,178.750,6.187,149.486
C01802=1128.223,-83.690,-46.457,178.747,6.186,149.486
C01803=1128.229,-83.940,-46.446,178.745,6.185,149.487
C01804=1128.234,-84.189,-46.437,178.743,6.185,149.487
C01805=1128.240,-84.439,-46.427,178.741,6.185,149.488
C01806=1128.245,-84.689,-46.418,178.739,6.184,149.488
C01807=1128.251,-84.938,-46.408,178.737,6.183,149.489
C01808=1128.256,-85.188,-46.399,178.735,6.182,149.489
C01809=1128.261,-85.438,-46.389,178.733,6.182,149.490
C01810=1128.267,-85.688,-46.380,178.730,6.182,149.490
C01811=1128.272,-85.937,-46.370,178.728,6.181,149.491
C01812=1128.277,-86.187,-46.361,178.726,6.181,149.491
C01813=1128.283,-86.438,-46.351,178.724,6.181,149.492
C01814=1128.287,-86.687,-46.342,178.722,6.180,149.492
C01815=1128.293,-86.937,-46.333,178.720,6.179,149.493
C01816=1128.298,-87.186,-46.322,178.718,6.179,149.493
C01817=1128.303,-87.436,-46.314,178.716,6.178,149.494
C01818=1128.309,-87.686,-46.304,178.714,6.178,149.494
C01819=1128.314,-87.936,-46.294,178.712,6.177,149.495
C01820=1128.320,-88.186,-46.285,178.710,6.177,149.495
C01821=1128.325,-88.436,-46.276,178.708,6.176,149.496
C01822=1128.330,-88.685,-46.266,178.706,6.175,149.496
C01823=1128.336,-88.935,-46.257,178.704,6.176,149.497
